C07313=1182.228,-66.696,-41.823,179.386,5.709,149.194
C07314=1182.223,-66.447,-41.834,179.389,5.710,149.194
C07315=1182.217,-66.196,-41.845,179.392,5.710,149.193
C07316=1182.213,-65.947,-41.856,179.393,5.710,149.192
C07317=1182.207,-65.697,-41.867,179.396,5.710,149.192
C07318=1182.202,-65.447,-41.878,179.398,5.711,149.191
C07319=1182.196,-65.198,-41.889,179.400,5.711,149.190
C07320=1182.191,-64.948,-41.900,179.403,5.711,149.190
C07321=1182.187,-64.698,-41.911,179.405,5.712,149.189
C07322=1182.181,-64.449,-41.921,179.407,5.712,149.189
C07323=1182.176,-64.199,-41.933,179.410,5.712,149.188
C07324=1182.171,-63.949,-41.945,179.412,5.713,149.187
C07325=1182.165,-63.700,-41.955,179.415,5.713,149.187
C07326=1182.161,-63.450,-41.966,179.417,5.713,149.186
C07327=1182.155,-63.200,-41.978,179.419,5.714,149.185
C07328=1182.150,-62.951,-41.988,179.422,5.714,149.185
C07329=1182.145,-62.701,-41.999,179.424,5.714,149.184
C07330=1182.139,-62.451,-42.011,179.426,5.715,149.184
C07331=1182.134,-62.201,-42.022,179.429,5.715,149.183
C07332=1182.129,-61.952,-42.033,179.431,5.715,149.182
C07333=1182.124,-61.702,-42.045,179.433,5.715,149.182
C07334=1182.118,-61.452,-42.055,179.436,5.716,149.181
C07335=1182.113,-61.203,-42.066,179.438,5.716,149.180
C07336=1182.108,-60.953,-42.078,179.440,5.716,149.180
C07337=1182.102,-60.703,-42.088,179.442,5.717,149.179
C07338=1182.098,-60.454,-42.100,179.445,5.717,149.178
C07339=1182.092,-60.204,-42.112,179.447,5.717,149.178
C07340=1182.087,-59.955,-42.122,179.449,5.718,149.177
C07341=1182.082,-59.705,-42.133,179.452,5.718,149.177
C07342=1182.077,-59.455,-42.145,179.454,5.718,149.176
C07343=1182.072,-59.205,-42.156,179.456,5.718,149.175
C07344=1182.067,-58.956,-42.167,179.459,5.719,149.175
C07345=1182.061,-58.705,-42.178,179.461,5.719,149.174
C07346=1182.056,-58.456,-42.190,179.463,5.719,149.173
C07347=1182.051,-58.206,-42.201,179.466,5.720,149.173
C07348=1182.045,-57.957,-42.212,179.468,5.721,149.172
C07349=1182.041,-57.707,-42.224,179.470,5.720,149.172
C07350=1182.035,-57.457,-42.235,179.473,5.721,149.171
C07351=1182.030,-57.208,-42.246,179.475,5.721,149.170
C07352=1182.024,-56.958,-42.258,179.477,5.721,149.170
C07353=1182.020,-56.708,-42.269,179.480,5.721,149.169
C07354=1182.015,-56.459,-42.280,179.482,5.722,149.169
C07355=1182.009,-56.209,-42.292,179.485,5.723,149.168
C07356=1182.004,-55.959,-42.302,179.487,5.722,149.167
C07357=1181.998,-55.709,-42.314,179.489,5.723,149.167
C07358=1181.994,-55.460,-42.325,179.492,5.724,149.166
C07359=1181.988,-55.210,-42.337,179.494,5.723,149.165
C07360=1181.983,-54.961,-42.348,179.496,5.724,149.165
C07361=1181.978,-54.711,-42.360,179.498,5.724,149.164
C07362=1181.973,-54.461,-42.371,179.501,5.725,149.163
C07363=1181.967,-54.211,-42.383,179.503,5.725,149.163
C07364=1181.963,-53.962,-42.395,179.505,5.725,149.162
C07365=1181.956,-53.712,-42.405,179.508,5.726,149.161
C07366=1181.952,-53.462,-42.417,179.511,5.726,149.161
C07367=1181.947,-53.213,-42.428,179.512,5.726,149.160
C07368=1181.942,-52.963,-42.440,179.515,5.727,149.160
C07369=1181.936,-52.713,-42.452,179.518,5.727,149.159
C07370=1181.931,-52.464,-42.463,179.519,5.727,149.158
C07371=1181.925,-52.214,-42.475,179.522,5.727,149.158
C07372=1181.921,-51.964,-42.486,179.525,5.728,149.157
C07373=1181.915,-51.714,-42.498,179.527,5.729,149.157
C07374=1181.911,-51.465,-42.509,179.529,5.728,149.156
C07375=1181.905,-51.215,-42.521,179.532,5.729,149.155
C07376=1181.900,-50.966,-42.532,179.534,5.730,149.155
C07377=1181.894,-50.716,-42.544,179.536,5.730,149.154
C07378=1181.890,-50.466,-42.555,179.538,5.730,149.153
C07379=1181.884,-50.216,-42.567,179.541,5.730,149.153
C07380=1181.878,-49.947,-42.580,179.543,5.731,149.152
C07381=1181.873,-49.676,-42.592,179.546,5.731,149.151
C07382=1181.868,-49.405,-42.605,179.549,5.732,149.151
C07383=1181.862,-49.136,-42.617,179.551,5.732,149.150
C07384=1181.857,-48.886,-42.629,179.553,5.732,149.149
C07385=1181.851,-48.636,-42.641,179.556,5.733,149.149
C07386=1181.846,-48.386,-42.652,179.558,5.733,149.148
C07387=1181.841,-48.137,-42.664,179.561,5.733,149.147
C07388=1181.836,-47.887,-42.676,179.562,5.733,149.147
C07389=1181.830,-47.637,-42.687,179.565,5.734,149.146
C07390=1181.825,-47.388,-42.698,179.568,5.734,149.145
C07391=1181.820,-47.138,-42.710,179.570,5.735,149.145
C07392=1181.815,-46.888,-42.722,179.572,5.735,149.144
C07393=1181.810,-46.639,-42.734,179.575,5.735,149.144
C07394=1181.805,-46.389,-42.746,179.577,5.736,149.143
C07395=1181.800,-46.139,-42.757,179.580,5.736,149.142
C07396=1181.794,-45.889,-42.769,179.582,5.737,149.142
C07397=1181.789,-45.639,-42.781,179.584,5.737,149.141
C07398=1181.784,-45.390,-42.792,179.587,5.737,149.141
C07399=1181.779,-45.141,-42.805,179.589,5.738,149.140
C07400=1181.773,-44.891,-42.817,179.592,5.738,149.139
C07401=1181.768,-44.642,-42.828,179.593,5.738,149.139
C07402=1181.763,-44.392,-42.840,179.596,5.739,149.138
C07403=1181.758,-44.142,-42.852,179.599,5.739,149.137
C07404=1181.752,-43.892,-42.864,179.601,5.740,149.137
C07405=1181.748,-43.643,-42.876,179.603,5.740,149.136
C07406=1181.742,-43.393,-42.887,179.606,5.740,149.135
C07407=1181.737,-43.143,-42.899,179.608,5.741,149.135
C07408=1181.732,-42.893,-42.911,179.611,5.741,149.134
C07409=1181.727,-42.644,-42.923,179.613,5.741,149.134
C07410=1181.722,-42.394,-42.935,179.615,5.741,149.133
C07411=1181.716,-42.144,-42.947,179.617,5.742,149.132
C07412=1181.712,-41.894,-42.958,179.620,5.743,149.132
C07413=1181.706,-41.645,-42.971,179.623,5.743,149.131
C07414=1181.701,-41.395,-42.983,179.624,5.743,149.130
C07415=1181.696,-41.145,-42.995,179.627,5.743,149.130
C07416=1181.691,-40.896,-43.007,179.630,5.744,149.129
C07417=1181.686,-40.646,-43.018,179.632,5.745,149.129
C07418=1181.680,-40.396,-43.030,179.635,5.745,149.128
C07419=1181.675,-40.147,-43.043,179.637,5.745,149.127
C07420=1181.670,-39.897,-43.055,179.639,5.745,149.126
C07421=1181.664,-39.648,-43.066,179.641,5.746,149.126
C07422=1181.659,-39.399,-43.078,179.644,5.746,149.125
C07423=1181.654,-39.149,-43.090,179.646,5.746,149.125
C07424=1181.648,-38.899,-43.102,179.648,5.747,149.124
C07425=1181.643,-38.650,-43.115,179.651,5.747,149.123
C07426=1181.639,-38.400,-43.126,179.654,5.748,149.123
C07427=1181.633,-38.150,-43.138,179.656,5.749,149.122
C07428=1181.628,-37.901,-43.151,179.658,5.748,149.122
C07429=1181.623,-37.650,-43.163,179.661,5.749,149.121
C07430=1181.618,-37.401,-43.175,179.663,5.750,149.120
C07431=1181.613,-37.151,-43.187,179.665,5.750,149.120
C07432=1181.608,-36.901,-43.199,179.668,5.750,149.119
C07433=1181.603,-36.652,-43.211,179.670,5.750,149.118
C07434=1181.597,-36.402,-43.223,179.672,5.751,149.118
C07435=1181.592,-36.153,-43.236,179.675,5.751,149.117
C07436=1181.587,-35.903,-43.248,179.678,5.752,149.116
C07437=1181.582,-35.653,-43.260,179.680,5.753,149.116
C07438=1181.576,-35.404,-43.272,179.682,5.752,149.115
C07439=1181.571,-35.154,-43.285,179.685,5.753,149.115
C07440=1181.566,-34.904,-43.296,179.687,5.753,149.114
C07441=1181.561,-34.655,-43.309,179.689,5.754,149.113
C07442=1181.556,-34.405,-43.320,179.692,5.754,149.113
C07443=1181.551,-34.156,-43.333,179.695,5.755,149.112
C07444=1181.545,-33.906,-43.345,179.696,5.755,149.112
C07445=1181.540,-33.657,-43.357,179.699,5.755,149.111
C07446=1181.535,-33.407,-43.369,179.702,5.756,149.110
C07447=1181.530,-33.158,-43.382,179.704,5.757,149.110
C07448=1181.525,-32.907,-43.394,179.707,5.757,149.109
C07449=1181.520,-32.658,-43.407,179.709,5.757,149.108
C07450=1181.514,-32.408,-43.419,179.711,5.757,149.108
C07451=1181.509,-32.158,-43.431,179.713,5.758,149.107
C07452=1181.504,-31.908,-43.443,179.716,5.758,149.106
C07453=1181.499,-31.659,-43.456,179.719,5.759,149.106
C07454=1181.494,-31.410,-43.468,179.721,5.760,149.105
C07455=1181.488,-31.160,-43.480,179.723,5.759,149.105
C07456=1181.483,-30.910,-43.493,179.726,5.760,149.104
C07457=1181.478,-30.660,-43.505,179.728,5.761,149.103
C07458=1181.473,-30.411,-43.518,179.731,5.761,149.103
C07459=1181.468,-30.161,-43.530,179.733,5.761,149.102
C07460=1181.463,-29.911,-43.542,179.735,5.762,149.101
C07461=1181.457,-29.662,-43.555,179.737,5.762,149.101
C07462=1181.452,-29.413,-43.567,179.740,5.762,149.100
C07463=1181.447,-29.163,-43.579,179.743,5.763,149.099
C07464=1181.442,-28.913,-43.592,179.745,5.764,149.099
C07465=1181.437,-28.663,-43.605,179.748,5.764,149.098
C07466=1181.432,-28.413,-43.617,179.750,5.764,149.098
C07467=1181.427,-28.164,-43.629,179.752,5.765,149.097
C07468=1181.422,-27.915,-43.642,179.755,5.765,149.096
C07469=1181.416,-27.665,-43.654,179.757,5.765,149.096
C07470=1181.412,-27.415,-43.667,179.759,5.766,149.095
C07471=1181.406,-27.166,-43.679,179.762,5.767,149.094
C07472=1181.401,-26.916,-43.692,179.765,5.767,149.094
C07473=1181.396,-26.666,-43.704,179.767,5.767,149.093
C07474=1181.391,-26.417,-43.716,179.769,5.768,149.093
C07475=1181.386,-26.168,-43.729,179.772,5.768,149.092
C07476=1181.381,-25.918,-43.742,179.774,5.769,149.091
C07477=1181.375,-25.667,-43.755,179.776,5.769,149.091
C07478=1181.370,-25.418,-43.767,179.779,5.770,149.090
C07479=1181.365,-25.169,-43.780,179.782,5.770,149.089
C07480=1181.360,-24.919,-43.792,179.783,5.770,149.089
C07481=1181.355,-24.669,-43.805,179.786,5.771,149.088
C07482=1181.350,-24.419,-43.817,179.789,5.771,149.087
C07483=1181.345,-24.170,-43.830,179.791,5.772,149.087
C07484=1181.339,-23.900,-43.844,179.794,5.772,149.086
C07485=1181.333,-23.631,-43.857,179.796,5.773,149.086
C07486=1181.328,-23.361,-43.871,179.799,5.773,149.085
C07487=1181.322,-23.091,-43.885,179.801,5.774,149.084
C07488=1181.317,-22.841,-43.897,179.804,5.774,149.084
C07489=1181.312,-22.592,-43.910,179.807,5.775,149.083
C07490=1181.307,-22.343,-43.922,179.809,5.776,149.082
C07491=1181.301,-22.092,-43.936,179.812,5.776,149.082
C07492=1181.296,-21.843,-43.949,179.814,5.776,149.081
C07493=1181.291,-21.594,-43.961,179.816,5.776,149.081
C07494=1181.286,-21.344,-43.974,179.819,5.777,149.080
C07495=1181.282,-21.094,-43.987,179.821,5.777,149.079
C07496=1181.275,-20.844,-43.999,179.824,5.778,149.078
C07497=1181.270,-20.595,-44.012,179.826,5.779,149.078
C07498=1181.266,-20.345,-44.025,179.829,5.779,149.077
C07499=1181.261,-20.096,-44.037,179.831,5.780,149.077
C07500=1181.255,-19.846,-44.051,179.833,5.780,149.076
C07501=1181.250,-19.597,-44.063,179.836,5.780,149.075
C07502=1181.245,-19.347,-44.076,179.838,5.781,149.075
C07503=1181.240,-19.097,-44.089,179.841,5.781,149.074
C07504=1181.234,-18.848,-44.102,179.843,5.782,149.074
C07505=1181.230,-18.598,-44.115,179.846,5.782,149.073
C07506=1181.225,-18.348,-44.128,179.848,5.783,149.072
C07507=1181.219,-18.099,-44.140,179.851,5.784,149.072
C07508=1181.214,-17.849,-44.153,179.853,5.783,149.071
C07509=1181.209,-17.599,-44.166,179.855,5.784,149.070
C07510=1181.204,-17.350,-44.179,179.858,5.784,149.070
C07511=1181.199,-17.101,-44.191,179.860,5.785,149.069
C07512=1181.194,-16.850,-44.205,179.863,5.785,149.068
C07513=1181.188,-16.601,-44.218,179.865,5.786,149.068
C07514=1181.183,-16.352,-44.230,179.868,5.787,149.067
C07515=1181.178,-16.101,-44.244,179.870,5.787,149.067
C07516=1181.173,-15.852,-44.256,179.873,5.788,149.066
C07517=1181.168,-15.603,-44.270,179.875,5.788,149.065
C07518=1181.163,-15.353,-44.283,179.877,5.788,149.065
C07519=1181.158,-15.104,-44.296,179.880,5.789,149.064
C07520=1181.153,-14.854,-44.309,179.882,5.789,149.064
C07521=1181.147,-14.604,-44.322,179.885,5.790,149.063
C07522=1181.142,-14.355,-44.335,179.887,5.790,149.062
C07523=1181.138,-14.105,-44.348,179.890,5.791,149.062
C07524=1181.132,-13.855,-44.361,179.892,5.792,149.061
C07525=1181.127,-13.606,-44.374,179.895,5.792,149.060
C07526=1181.122,-13.356,-44.388,179.898,5.793,149.060
C07527=1181.117,-13.107,-44.400,179.900,5.793,149.059
C07528=1181.112,-12.857,-44.413,179.902,5.794,149.059
C07529=1181.106,-12.607,-44.426,179.904,5.793,149.058
C07530=1181.101,-12.358,-44.439,179.907,5.794,149.057
C07531=1181.097,-12.108,-44.453,179.909,5.795,149.057
C07532=1181.091,-11.859,-44.466,179.912,5.795,149.056
C07533=1181.086,-11.609,-44.479,179.915,5.796,149.055
C07534=1181.081,-11.359,-44.492,179.917,5.797,149.055
C07535=1181.076,-11.110,-44.505,179.919,5.797,149.054
C07536=1181.071,-10.860,-44.519,179.922,5.797,149.053
C07537=1181.065,-10.611,-44.532,179.924,5.798,149.053
C07538=1181.061,-10.361,-44.545,179.927,5.799,149.052
C07539=1181.055,-10.112,-44.558,179.930,5.799,149.052
C07540=1181.051,-9.862,-44.571,179.932,5.800,149.051
C07541=1181.045,-9.612,-44.585,179.934,5.800,149.050
C07542=1181.040,-9.363,-44.597,179.936,5.800,149.050
C07543=1181.035,-9.113,-44.612,179.939,5.801,149.049
C07544=1181.030,-8.864,-44.624,179.941,5.801,149.049
C07545=1181.024,-8.613,-44.638,179.944,5.802,149.048
C07546=1181.020,-8.365,-44.651,179.947,5.802,149.047
C07547=1181.014,-8.114,-44.665,179.949,5.803,149.047
C07548=1181.009,-7.865,-44.677,179.951,5.804,149.046
C07549=1181.004,-7.615,-44.691,179.954,5.804,149.045
C07550=1180.999,-7.366,-44.704,179.956,5.805,149.045
C07551=1180.994,-7.116,-44.718,179.959,5.805,149.044
C07552=1180.989,-6.867,-44.731,179.962,5.806,149.043
C07553=1180.984,-6.617,-44.744,179.964,5.806,149.043
C07554=1180.979,-6.367,-44.757,179.966,5.807,149.042
C07555=1180.974,-6.118,-44.771,179.969,5.808,149.042
C07556=1180.969,-5.868,-44.784,179.972,5.808,149.041
C07557=1180.964,-5.619,-44.798,179.974,5.809,149.040
C07558=1180.959,-5.369,-44.811,179.977,5.809,149.040
C07559=1180.953,-5.119,-44.824,179.979,5.810,149.039
C07560=1180.948,-4.870,-44.838,179.981,5.810,149.039
C07561=1180.943,-4.620,-44.851,179.983,5.810,149.038
C07562=1180.938,-4.371,-44.865,179.986,5.811,149.037
C07563=1180.933,-4.121,-44.878,179.989,5.811,149.037
C07564=1180.928,-3.872,-44.892,179.991,5.812,149.036
C07565=1180.922,-3.622,-44.906,179.994,5.813,149.035
C07566=1180.918,-3.373,-44.919,179.996,5.813,149.035
C07567=1180.912,-3.123,-44.932,179.998,5.814,149.034
C07568=1180.907,-2.874,-44.946,-179.999,5.814,149.034
C07569=1180.902,-2.624,-44.959,-179.996,5.815,149.033
C07570=1180.897,-2.375,-44.973,-179.994,5.816,149.032
C07571=1180.892,-2.125,-44.986,-179.992,5.816,149.032
C07572=1180.887,-1.875,-45.001,-179.989,5.817,149.031
C07573=1180.881,-1.625,-45.014,-179.986,5.817,149.030
C07574=1180.877,-1.376,-45.027,-179.984,5.818,149.030
C07575=1180.871,-1.126,-45.041,-179.981,5.818,149.029
C07576=1180.866,-0.876,-45.055,-179.979,5.819,149.029
C07577=1180.861,-0.627,-45.067,-179.977,5.820,149.028
C07578=1180.856,-0.377,-45.082,-179.974,5.820,149.027
C07579=1180.851,-0.128,-45.096,-179.971,5.821,149.027
C07580=1180.846,0.122,-45.109,-179.969,5.822,149.026
C07581=1180.841,0.371,-45.123,-179.966,5.822,149.026
C07582=1180.835,0.621,-45.136,-179.964,5.823,149.025
C07583=1180.831,0.870,-45.150,-179.962,5.823,149.024
C07584=1180.826,1.119,-45.164,-179.959,5.824,149.024
C07585=1180.820,1.370,-45.177,-179.956,5.824,149.023
C07586=1180.815,1.619,-45.192,-179.954,5.825,149.022
C07587=1180.810,1.868,-45.205,-179.951,5.826,149.022
C07588=1180.805,2.138,-45.220,-179.949,5.826,149.021
C07589=1180.800,2.407,-45.235,-179.946,5.827,149.020
C07590=1180.794,2.676,-45.250,-179.943,5.827,149.020
C07591=1180.788,2.945,-45.264,-179.941,5.828,149.019
C07592=1180.783,3.195,-45.278,-179.938,5.828,149.018
C07593=1180.779,3.445,-45.292,-179.936,5.829,149.018
C07594=1180.773,3.694,-45.306,-179.933,5.829,149.017
C07595=1180.768,3.944,-45.319,-179.931,5.830,149.017
C07596=1180.763,4.194,-45.333,-179.929,5.831,149.016
C07597=1180.758,4.443,-45.347,-179.926,5.831,149.015
C07598=1180.753,4.692,-45.361,-179.923,5.832,149.015
C07599=1180.748,4.943,-45.375,-179.921,5.832,149.014
C07600=1180.742,5.192,-45.389,-179.918,5.833,149.014
C07601=1180.737,5.441,-45.403,-179.916,5.833,149.013
C07602=1180.733,5.691,-45.416,-179.914,5.834,149.012
C07603=1180.727,5.940,-45.430,-179.911,5.835,149.012
C07604=1180.722,6.190,-45.444,-179.908,5.835,149.011
C07605=1180.717,6.440,-45.458,-179.906,5.836,149.011
C07606=1180.712,6.689,-45.472,-179.903,5.836,149.010
C07607=1180.707,6.938,-45.486,-179.901,5.837,149.009
C07608=1180.703,7.188,-45.500,-179.898,5.837,149.009
C07609=1180.697,7.437,-45.513,-179.896,5.838,149.008
C07610=1180.692,7.687,-45.528,-179.893,5.840,149.007
C07611=1180.687,7.937,-45.542,-179.890,5.840,149.007
C07612=1180.682,8.187,-45.556,-179.888,5.841,149.006
C07613=1180.676,8.436,-45.570,-179.885,5.841,149.006
C07614=1180.671,8.685,-45.584,-179.883,5.842,149.005
C07615=1180.666,8.935,-45.599,-179.880,5.843,149.004
C07616=1180.661,9.184,-45.611,-179.878,5.843,149.004
C07617=1180.656,9.434,-45.625,-179.875,5.844,149.003
C07618=1180.651,9.684,-45.640,-179.873,5.845,149.003
C07619=1180.646,9.934,-45.654,-179.870,5.845,149.002
C07620=1180.641,10.183,-45.668,-179.868,5.845,149.001
C07621=1180.636,10.432,-45.682,-179.866,5.846,149.001
C07622=1180.631,10.682,-45.696,-179.863,5.847,149.000
C07623=1180.626,10.932,-45.711,-179.860,5.847,148.999
C07624=1180.620,11.181,-45.725,-179.858,5.848,148.999
C07625=1180.616,11.430,-45.739,-179.855,5.849,148.998
C07626=1180.611,11.680,-45.753,-179.853,5.849,148.998
C07627=1180.606,11.930,-45.767,-179.851,5.850,148.997
C07628=1180.601,12.179,-45.782,-179.848,5.850,148.996
C07629=1180.595,12.428,-45.796,-179.845,5.851,148.996
C07630=1180.590,12.678,-45.810,-179.843,5.851,148.995
C07631=1180.585,12.928,-45.824,-179.840,5.852,148.995
C07632=1180.580,13.178,-45.839,-179.838,5.853,148.994
C07633=1180.575,13.427,-45.852,-179.835,5.853,148.993
C07634=1180.570,13.676,-45.867,-179.833,5.854,148.993
C07635=1180.565,13.926,-45.881,-179.830,5.855,148.992
C07636=1180.560,14.176,-45.895,-179.828,5.855,148.991
C07637=1180.555,14.425,-45.910,-179.825,5.857,148.991
C07638=1180.549,14.674,-45.923,-179.822,5.857,148.990
C07639=1180.544,14.924,-45.938,-179.820,5.858,148.990
C07640=1180.540,15.173,-45.953,-179.817,5.858,148.989
C07641=1180.535,15.423,-45.967,-179.815,5.859,148.988
C07642=1180.530,15.673,-45.981,-179.812,5.859,148.988
C07643=1180.525,15.922,-45.996,-179.810,5.860,148.987
C07644=1180.519,16.171,-46.009,-179.807,5.861,148.987
C07645=1180.514,16.421,-46.024,-179.805,5.861,148.986
C07646=1180.509,16.671,-46.038,-179.803,5.862,148.986
C07647=1180.504,16.921,-46.052,-179.800,5.863,148.985
C07648=1180.500,17.170,-46.067,-179.797,5.863,148.984
C07649=1180.494,17.420,-46.082,-179.795,5.864,148.984
C07650=1180.489,17.669,-46.096,-179.792,5.864,148.983
C07651=1180.484,17.918,-46.110,-179.790,5.865,148.982
C07652=1180.479,18.168,-46.125,-179.787,5.867,148.982
C07653=1180.474,18.417,-46.140,-179.784,5.867,148.981
C07654=1180.469,18.667,-46.154,-179.782,5.868,148.981
C07655=1180.464,18.917,-46.168,-179.780,5.868,148.980
C07656=1180.459,19.166,-46.182,-179.777,5.869,148.979
C07657=1180.454,19.416,-46.197,-179.774,5.869,148.979
C07658=1180.449,19.665,-46.212,-179.772,5.870,148.978
C07659=1180.444,19.915,-46.227,-179.769,5.871,148.978
C07660=1180.438,20.164,-46.241,-179.767,5.871,148.977
C07661=1180.434,20.413,-46.255,-179.765,5.872,148.976
C07662=1180.429,20.663,-46.270,-179.762,5.873,148.976
C07663=1180.424,20.913,-46.284,-179.759,5.873,148.975
C07664=1180.418,21.163,-46.299,-179.757,5.875,148.975
C07665=1180.413,21.412,-46.314,-179.754,5.875,148.974
C07666=1180.408,21.662,-46.328,-179.751,5.876,148.973
C07667=1180.403,21.911,-46.342,-179.749,5.877,148.973
C07668=1180.399,22.160,-46.357,-179.747,5.877,148.972
C07669=1180.393,22.410,-46.372,-179.744,5.878,148.971
C07670=1180.388,22.660,-46.387,-179.742,5.878,148.971
C07671=1180.383,22.909,-46.402,-179.739,5.879,148.970
C07672=1180.379,23.159,-46.416,-179.736,5.879,148.970
C07673=1180.373,23.409,-46.431,-179.734,5.880,148.969
C07674=1180.368,23.657,-46.445,-179.731,5.882,148.968
C07675=1180.363,23.907,-46.460,-179.728,5.882,148.968
C07676=1180.358,24.156,-46.475,-179.726,5.883,148.967
C07677=1180.352,24.406,-46.490,-179.724,5.883,148.967
C07678=1180.348,24.655,-46.505,-179.721,5.884,148.966
C07679=1180.343,24.905,-46.519,-179.719,5.885,148.966
C07680=1180.338,25.155,-46.533,-179.716,5.885,148.965
C07681=1180.332,25.404,-46.549,-179.714,5.886,148.964
C07682=1180.327,25.654,-46.563,-179.711,5.887,148.964
C07683=1180.323,25.903,-46.578,-179.708,5.888,148.963
C07684=1180.317,26.153,-46.593,-179.706,5.889,148.963
C07685=1180.312,26.402,-46.608,-179.703,5.889,148.962
C07686=1180.307,26.652,-46.622,-179.701,5.890,148.961
C07687=1180.302,26.901,-46.638,-179.698,5.891,148.961
C07688=1180.297,27.151,-46.652,-179.696,5.891,148.960
C07689=1180.292,27.400,-46.667,-179.693,5.892,148.959
C07690=1180.287,27.650,-46.682,-179.691,5.892,148.959
C07691=1180.282,27.899,-46.697,-179.688,5.894,148.958
C07692=1180.277,28.168,-46.713,-179.685,5.894,148.958
C07693=1180.271,28.437,-46.729,-179.682,5.895,148.957
C07694=1180.266,28.706,-46.745,-179.679,5.896,148.956
C07695=1180.260,28.975,-46.761,-179.677,5.897,148.956
C07696=1180.255,29.224,-46.776,-179.674,5.897,148.955
C07697=1180.251,29.473,-46.791,-179.672,5.898,148.954
C07698=1180.245,29.723,-46.806,-179.670,5.899,148.954
C07699=1180.241,29.972,-46.821,-179.667,5.899,148.953
C07700=1180.235,30.223,-46.836,-179.664,5.900,148.953
C07701=1180.231,30.472,-46.851,-179.662,5.901,148.952
C07702=1180.226,30.721,-46.866,-179.659,5.902,148.952
C07703=1180.220,30.971,-46.881,-179.656,5.902,148.951
C07704=1180.216,31.220,-46.896,-179.654,5.903,148.950
C07705=1180.210,31.469,-46.911,-179.652,5.904,148.950
C07706=1180.205,31.719,-46.926,-179.649,5.905,148.949
C07707=1180.200,31.969,-46.941,-179.646,5.906,148.949
C07708=1180.195,32.218,-46.956,-179.643,5.906,148.948
C07709=1180.190,32.468,-46.971,-179.641,5.907,148.947
C07710=1180.185,32.717,-46.986,-179.639,5.908,148.947
C07711=1180.181,32.967,-47.001,-179.636,5.908,148.946
C07712=1180.175,33.217,-47.016,-179.634,5.909,148.946
C07713=1180.171,33.466,-47.031,-179.631,5.910,148.945
C07714=1180.165,33.715,-47.047,-179.628,5.911,148.944
C07715=1180.161,33.964,-47.062,-179.626,5.912,148.944
C07716=1180.155,34.214,-47.077,-179.623,5.912,148.943
C07717=1180.150,34.463,-47.092,-179.621,5.913,148.943
C07718=1180.145,34.713,-47.107,-179.618,5.914,148.942
C07719=1180.140,34.963,-47.123,-179.615,5.915,148.941
C07720=1180.135,35.212,-47.138,-179.613,5.916,148.941
C07721=1180.130,35.462,-47.153,-179.610,5.916,148.940
C07722=1180.125,35.711,-47.168,-179.608,5.917,148.940
C07723=1180.120,35.960,-47.184,-179.606,5.918,148.939
C07724=1180.115,36.209,-47.199,-179.603,5.918,148.938
C07725=1180.110,36.459,-47.214,-179.600,5.919,148.938
C07726=1180.105,36.709,-47.229,-179.598,5.920,148.937
C07727=1180.100,36.959,-47.245,-179.595,5.921,148.937
C07728=1180.095,37.208,-47.260,-179.593,5.922,148.936
C07729=1180.090,37.457,-47.275,-179.590,5.922,148.936
C07730=1180.085,37.707,-47.291,-179.587,5.923,148.935
C07731=1180.080,37.956,-47.306,-179.585,5.924,148.934
C07732=1180.075,38.206,-47.322,-179.582,5.925,148.934
C07733=1180.070,38.455,-47.337,-179.579,5.925,148.933
C07734=1180.065,38.705,-47.352,-179.577,5.926,148.933
C07735=1180.059,38.954,-47.367,-179.575,5.927,148.932
C07736=1180.055,39.203,-47.382,-179.572,5.928,148.932
C07737=1180.050,39.453,-47.398,-179.569,5.929,148.931
C07738=1180.045,39.703,-47.414,-179.567,5.929,148.930
C07739=1180.040,39.952,-47.429,-179.564,5.930,148.930
C07740=1180.035,40.201,-47.444,-179.562,5.931,148.929
C07741=1180.030,40.451,-47.460,-179.559,5.932,148.929
C07742=1180.025,40.701,-47.475,-179.556,5.933,148.928
C07743=1180.020,40.950,-47.491,-179.554,5.933,148.927
C07744=1180.014,41.199,-47.506,-179.552,5.934,148.927
C07745=1180.010,41.448,-47.521,-179.549,5.935,148.926
C07746=1180.005,41.699,-47.537,-179.546,5.936,148.926
C07747=1179.999,41.948,-47.553,-179.544,5.937,148.925
C07748=1179.995,42.197,-47.568,-179.541,5.938,148.924
C07749=1179.990,42.447,-47.584,-179.539,5.938,148.924
C07750=1179.985,42.697,-47.599,-179.536,5.940,148.923
C07751=1179.979,42.946,-47.615,-179.533,5.940,148.923
C07752=1179.975,43.195,-47.630,-179.531,5.941,148.922
C07753=1179.970,43.445,-47.646,-179.528,5.942,148.921
C07754=1179.965,43.694,-47.662,-179.526,5.943,148.921
C07755=1179.959,43.943,-47.678,-179.523,5.944,148.920
C07756=1179.955,44.192,-47.693,-179.520,5.944,148.920
C07757=1179.950,44.443,-47.709,-179.518,5.945,148.919
C07758=1179.945,44.692,-47.724,-179.515,5.946,148.919
C07759=1179.939,44.941,-47.740,-179.513,5.947,148.918
C07760=1179.935,45.191,-47.755,-179.510,5.948,148.917
C07761=1179.930,45.441,-47.771,-179.507,5.948,148.917
C07762=1179.925,45.689,-47.787,-179.505,5.949,148.916
C07763=1179.920,45.939,-47.803,-179.503,5.950,148.916
C07764=1179.914,46.189,-47.819,-179.499,5.951,148.915
C07765=1179.910,46.438,-47.834,-179.497,5.952,148.915
C07766=1179.905,46.688,-47.850,-179.495,5.952,148.914
C07767=1179.900,46.937,-47.866,-179.492,5.953,148.913
C07768=1179.895,47.186,-47.882,-179.489,5.955,148.913
C07769=1179.890,47.436,-47.898,-179.486,5.955,148.912
C07770=1179.885,47.685,-47.913,-179.484,5.956,148.912
C07771=1179.880,47.934,-47.929,-179.482,5.957,148.911
C07772=1179.875,48.184,-47.945,-179.479,5.958,148.911
C07773=1179.870,48.434,-47.960,-179.476,5.959,148.910
C07774=1179.864,48.683,-47.976,-179.474,5.960,148.909
C07775=1179.860,48.933,-47.993,-179.472,5.960,148.909
C07776=1179.855,49.182,-48.008,-179.468,5.961,148.908
C07777=1179.851,49.432,-48.024,-179.466,5.962,148.908
C07778=1179.845,49.681,-48.039,-179.464,5.963,148.907
C07779=1179.840,49.930,-48.055,-179.461,5.964,148.907
C07780=1179.835,50.180,-48.071,-179.458,5.965,148.906
C07781=1179.830,50.429,-48.087,-179.456,5.966,148.905
C07782=1179.825,50.679,-48.104,-179.453,5.966,148.905
C07783=1179.820,50.928,-48.119,-179.451,5.967,148.904
C07784=1179.815,51.177,-48.136,-179.448,5.969,148.904
C07785=1179.810,51.427,-48.152,-179.445,5.969,148.903
C07786=1179.805,51.677,-48.167,-179.443,5.970,148.902
C07787=1179.800,51.926,-48.184,-179.440,5.971,148.902
C07788=1179.795,52.176,-48.199,-179.437,5.972,148.901
C07789=1179.791,52.424,-48.215,-179.435,5.973,148.901
C07790=1179.786,52.674,-48.231,-179.433,5.973,148.900
C07791=1179.780,52.924,-48.247,-179.430,5.975,148.900
C07792=1179.776,53.173,-48.263,-179.427,5.975,148.899
C07793=1179.771,53.422,-48.279,-179.425,5.976,148.898
C07794=1179.766,53.672,-48.296,-179.422,5.977,148.898
C07795=1179.761,53.921,-48.311,-179.419,5.978,148.897
C07796=1179.755,54.190,-48.328,-179.417,5.979,148.897
C07797=1179.750,54.459,-48.347,-179.414,5.980,148.896
C07798=1179.744,54.727,-48.364,-179.411,5.981,148.895
C07799=1179.739,54.996,-48.381,-179.408,5.982,148.895
C07800=1179.734,55.245,-48.398,-179.406,5.983,148.894
C07801=1179.729,55.494,-48.413,-179.403,5.984,148.894
C07802=1179.724,55.744,-48.430,-179.401,5.984,148.893
C07803=1179.719,55.993,-48.445,-179.398,5.986,148.893
C07804=1179.714,56.243,-48.462,-179.395,5.986,148.892
C07805=1179.709,56.492,-48.478,-179.393,5.987,148.892
C07806=1179.705,56.742,-48.494,-179.390,5.989,148.891
C07807=1179.699,56.991,-48.511,-179.388,5.989,148.890
C07808=1179.695,57.241,-48.527,-179.385,5.990,148.890
C07809=1179.690,57.489,-48.543,-179.382,5.991,148.889
C07810=1179.685,57.740,-48.559,-179.380,5.992,148.889
C07811=1179.679,57.989,-48.576,-179.377,5.993,148.888
C07812=1179.675,58.238,-48.592,-179.375,5.994,148.888
C07813=1179.669,58.487,-48.608,-179.372,5.995,148.887
C07814=1179.665,58.737,-48.625,-179.369,5.996,148.886
C07815=1179.659,58.986,-48.640,-179.367,5.996,148.886
C07816=1179.655,59.236,-48.657,-179.364,5.998,148.885
C07817=1179.650,59.485,-48.673,-179.361,5.998,148.885
C07818=1179.645,59.735,-48.689,-179.359,5.999,148.884
C07819=1179.639,59.984,-48.706,-179.356,6.001,148.884
C07820=1179.635,60.233,-48.723,-179.353,6.001,148.883
C07821=1179.630,60.483,-48.739,-179.351,6.002,148.882
C07822=1179.625,60.732,-48.755,-179.348,6.003,148.882
C07823=1179.620,60.982,-48.772,-179.346,6.004,148.881
C07824=1179.615,61.230,-48.788,-179.343,6.005,148.881
C07825=1179.610,61.481,-48.805,-179.341,6.007,148.880
C07826=1179.605,61.730,-48.821,-179.338,6.007,148.880
C07827=1179.600,61.979,-48.837,-179.335,6.008,148.879
C07828=1179.596,62.229,-48.854,-179.333,6.009,148.879
C07829=1179.590,62.478,-48.870,-179.330,6.010,148.878
C07830=1179.585,62.728,-48.887,-179.328,6.011,148.877
C07831=1179.580,62.977,-48.903,-179.325,6.012,148.877
C07832=1179.575,63.226,-48.920,-179.322,6.013,148.876
C07833=1179.571,63.476,-48.937,-179.320,6.013,148.876
C07834=1179.565,63.725,-48.953,-179.317,6.015,148.875
C07835=1179.560,63.975,-48.970,-179.314,6.016,148.875
C07836=1179.556,64.224,-48.986,-179.312,6.017,148.874
C07837=1179.551,64.473,-49.002,-179.309,6.018,148.873
C07838=1179.546,64.723,-49.020,-179.306,6.018,148.873
C07839=1179.541,64.972,-49.036,-179.304,6.019,148.872
C07840=1179.536,65.221,-49.053,-179.301,6.021,148.872
C07841=1179.531,65.471,-49.070,-179.299,6.021,148.871
C07842=1179.525,65.720,-49.086,-179.296,6.022,148.871
C07843=1179.521,65.970,-49.102,-179.294,6.024,148.870
C07844=1179.516,66.219,-49.119,-179.291,6.024,148.870
C07845=1179.511,66.468,-49.136,-179.288,6.026,148.869
C07846=1179.506,66.718,-49.152,-179.286,6.026,148.868
C07847=1179.502,66.967,-49.169,-179.283,6.027,148.868
C07848=1179.496,67.216,-49.186,-179.280,6.029,148.867
C07849=1179.491,67.466,-49.203,-179.278,6.030,148.867
C07850=1179.487,67.715,-49.219,-179.275,6.030,148.866
C07851=1179.482,67.965,-49.237,-179.273,6.032,148.866
C07852=1179.477,68.214,-49.253,-179.270,6.032,148.865
C07853=1179.471,68.464,-49.270,-179.268,6.033,148.865
C07854=1179.467,68.713,-49.287,-179.265,6.035,148.864
C07855=1179.462,68.962,-49.303,-179.262,6.035,148.863
C07856=1179.457,69.212,-49.320,-179.259,6.037,148.863
C07857=1179.452,69.461,-49.337,-179.257,6.037,148.862
C07858=1179.448,69.711,-49.354,-179.255,6.038,148.862
C07859=1179.442,69.960,-49.371,-179.251,6.040,148.861
C07860=1179.437,70.209,-49.387,-179.249,6.040,148.861
C07861=1179.432,70.459,-49.405,-179.247,6.041,148.860
C07862=1179.427,70.708,-49.421,-179.244,6.043,148.860
C07863=1179.422,70.958,-49.438,-179.241,6.043,148.859
C07864=1179.418,71.207,-49.456,-179.238,6.045,148.859
C07865=1179.413,71.456,-49.472,-179.236,6.045,148.858
C07866=1179.407,71.705,-49.489,-179.234,6.046,148.858
C07867=1179.403,71.955,-49.506,-179.231,6.048,148.857
C07868=1179.398,72.204,-49.523,-179.228,6.049,148.856
C07869=1179.393,72.454,-49.540,-179.225,6.050,148.856
C07870=1179.387,72.703,-49.557,-179.223,6.051,148.855
C07871=1179.383,72.952,-49.574,-179.220,6.051,148.855
C07872=1179.378,73.202,-49.591,-179.218,6.053,148.854
C07873=1179.374,73.451,-49.608,-179.215,6.054,148.854
C07874=1179.368,73.701,-49.625,-179.212,6.055,148.853
C07875=1179.363,73.950,-49.642,-179.210,6.056,148.853
C07876=1179.358,74.199,-49.660,-179.208,6.057,148.852
C07877=1179.354,74.448,-49.676,-179.204,6.058,148.851
C07878=1179.349,74.698,-49.693,-179.202,6.059,148.851
C07879=1179.344,74.948,-49.710,-179.199,6.060,148.850
C07880=1179.339,75.196,-49.728,-179.197,6.061,148.850
C07881=1179.333,75.446,-49.745,-179.194,6.062,148.849
C07882=1179.329,75.695,-49.762,-179.191,6.063,148.849
C07883=1179.324,75.945,-49.779,-179.189,6.064,148.848
C07884=1179.320,76.194,-49.796,-179.186,6.066,148.848
C07885=1179.314,76.444,-49.814,-179.183,6.066,148.847
C07886=1179.309,76.693,-49.830,-179.181,6.068,148.847
C07887=1179.304,76.942,-49.848,-179.178,6.068,148.846
C07888=1179.299,77.192,-49.865,-179.176,6.069,148.846
C07889=1179.295,77.441,-49.882,-179.173,6.071,148.845
C07890=1179.290,77.690,-49.900,-179.171,6.071,148.845
C07891=1179.285,77.940,-49.916,-179.167,6.073,148.844
C07892=1179.279,78.189,-49.933,-179.165,6.074,148.843
C07893=1179.274,78.438,-49.951,-179.162,6.075,148.843
C07894=1179.270,78.688,-49.968,-179.160,6.076,148.842
C07895=1179.265,78.937,-49.986,-179.157,6.077,148.842
C07896=1179.260,79.187,-50.003,-179.155,6.078,148.841
C07897=1179.255,79.436,-50.020,-179.152,6.079,148.841
C07898=1179.250,79.685,-50.038,-179.149,6.080,148.840
C07899=1179.245,79.935,-50.055,-179.147,6.081,148.840
C07900=1179.240,80.202,-50.074,-179.144,6.083,148.839
C07901=1179.235,80.471,-50.092,-179.141,6.083,148.838
C07902=1179.230,80.740,-50.111,-179.138,6.085,148.838
C07903=1179.224,81.008,-50.130,-179.135,6.086,148.837
C07904=1179.219,81.257,-50.147,-179.133,6.087,148.837
C07905=1179.214,81.506,-50.165,-179.130,6.089,148.836
C07906=1179.209,81.756,-50.182,-179.127,6.089,148.836
C07907=1179.204,82.005,-50.200,-179.125,6.091,148.835
C07908=1179.200,82.255,-50.217,-179.122,6.091,148.835
C07909=1179.195,82.504,-50.235,-179.120,6.092,148.834
C07910=1179.190,82.754,-50.252,-179.117,6.094,148.834
C07911=1179.185,83.003,-50.270,-179.114,6.094,148.833
C07912=1179.180,83.252,-50.286,-179.112,6.096,148.833
C07913=1179.175,83.501,-50.304,-179.109,6.097,148.832
C07914=1179.171,83.751,-50.322,-179.106,6.098,148.832
C07915=1179.165,84.000,-50.340,-179.104,6.099,148.831
C07916=1179.160,84.250,-50.358,-179.101,6.101,148.831
C07917=1179.156,84.499,-50.374,-179.098,6.101,148.830
C07918=1179.151,84.748,-50.392,-179.096,6.103,148.829
C07919=1179.146,84.997,-50.410,-179.093,6.103,148.829
C07920=1179.141,85.247,-50.428,-179.090,6.105,148.828
C07921=1179.136,85.496,-50.446,-179.088,6.106,148.828
C07922=1179.132,85.745,-50.463,-179.085,6.107,148.827
C07923=1179.127,85.995,-50.480,-179.083,6.108,148.827
C07924=1179.122,86.244,-50.498,-179.080,6.110,148.826
C07925=1179.117,86.493,-50.516,-179.078,6.111,148.826
C07926=1179.112,86.743,-50.533,-179.075,6.111,148.825
C07927=1179.107,86.992,-50.551,-179.072,6.113,148.825
C07928=1179.102,87.242,-50.569,-179.070,6.113,148.824
C07929=1179.097,87.491,-50.586,-179.067,6.115,148.824
C07930=1179.092,87.740,-50.604,-179.065,6.116,148.823
C07931=1179.087,87.989,-50.622,-179.062,6.117,148.823
C07932=1179.082,88.239,-50.640,-179.059,6.118,148.822
C07933=1179.077,88.488,-50.657,-179.056,6.120,148.822
C07934=1179.072,88.738,-50.675,-179.054,6.121,148.821
C07935=1179.067,88.987,-50.693,-179.051,6.122,148.820
C07936=1179.063,89.236,-50.711,-179.049,6.123,148.820
C07937=1179.058,89.485,-50.729,-179.045,6.124,148.819
C07938=1179.052,89.735,-50.746,-179.043,6.125,148.819
C07939=1179.047,89.984,-50.764,-179.041,6.127,148.819
C07940=1179.043,90.233,-50.782,-179.038,6.127,148.818
C07941=1179.038,90.482,-50.800,-179.035,6.129,148.817
C07942=1179.034,90.732,-50.818,-179.033,6.130,148.817
C07943=1179.029,90.981,-50.836,-179.030,6.131,148.816
C07944=1179.024,91.230,-50.854,-179.027,6.133,148.816
C07945=1179.019,91.480,-50.871,-179.025,6.134,148.815
C07946=1179.014,91.729,-50.889,-179.022,6.135,148.815
C07947=1179.009,91.978,-50.907,-179.019,6.136,148.814
C07948=1179.004,92.228,-50.925,-179.017,6.137,148.814
C07949=1178.999,92.477,-50.943,-179.014,6.138,148.813
C07950=1178.994,92.726,-50.961,-179.011,6.140,148.813
C07951=1178.990,92.976,-50.980,-179.009,6.140,148.812
C07952=1178.985,93.225,-50.998,-179.006,6.142,148.812
C07953=1178.980,93.474,-51.016,-179.004,6.143,148.811
C07954=1178.975,93.723,-51.034,-179.001,6.144,148.811
C07955=1178.970,93.973,-51.052,-178.998,6.145,148.810
C07956=1178.965,94.222,-51.070,-178.995,6.147,148.810
C07957=1178.960,94.471,-51.088,-178.993,6.147,148.809
C07958=1178.955,94.720,-51.106,-178.990,6.149,148.809
C07959=1178.951,94.970,-51.124,-178.988,6.150,148.808
C07960=1178.946,95.219,-51.142,-178.985,6.151,148.808
C07961=1178.941,95.469,-51.160,-178.982,6.153,148.807
C07962=1178.936,95.718,-51.178,-178.980,6.154,148.807
C07963=1178.931,95.967,-51.196,-178.977,6.155,148.806
C07964=1178.926,96.216,-51.214,-178.974,6.156,148.806
C07965=1178.922,96.466,-51.233,-178.972,6.158,148.805
C07966=1178.916,96.716,-51.251,-178.969,6.158,148.805
C07967=1178.911,96.965,-51.269,-178.966,6.160,148.804
C07968=1178.906,97.214,-51.287,-178.964,6.161,148.804
C07969=1178.902,97.462,-51.306,-178.961,6.162,148.803
C07970=1178.897,97.712,-51.324,-178.959,6.163,148.803
C07971=1178.893,97.961,-51.342,-178.956,6.165,148.802
C07972=1178.888,98.211,-51.360,-178.953,6.166,148.802
C07973=1178.882,98.460,-51.379,-178.951,6.167,148.801
C07974=1178.878,98.710,-51.397,-178.948,6.169,148.801
C07975=1178.873,98.959,-51.416,-178.945,6.169,148.800
C07976=1178.868,99.208,-51.434,-178.942,6.171,148.799
C07977=1178.863,99.457,-51.452,-178.940,6.172,148.799
C07978=1178.858,99.706,-51.470,-178.937,6.173,148.799
C07979=1178.853,99.956,-51.489,-178.934,6.175,148.798
C07980=1178.849,100.205,-51.507,-178.932,6.176,148.798
C07981=1178.844,100.454,-51.525,-178.929,6.177,148.797
C07982=1178.839,100.703,-51.543,-178.927,6.178,148.797
C07983=1178.834,100.953,-51.562,-178.924,6.180,148.796
C07984=1178.829,101.202,-51.581,-178.921,6.180,148.795
C07985=1178.824,101.451,-51.599,-178.919,6.182,148.795
C07986=1178.820,101.701,-51.617,-178.916,6.184,148.795
C07987=1178.815,101.950,-51.637,-178.913,6.184,148.794
C07988=1178.810,102.199,-51.655,-178.911,6.186,148.794
C07989=1178.805,102.448,-51.673,-178.908,6.187,148.793
C07990=1178.800,102.698,-51.691,-178.905,6.188,148.793
C07991=1178.795,102.947,-51.710,-178.903,6.190,148.792
C07992=1178.790,103.196,-51.728,-178.900,6.191,148.791
C07993=1178.786,103.446,-51.748,-178.897,6.192,148.791
C07994=1178.781,103.695,-51.766,-178.895,6.193,148.791
C07995=1178.776,103.944,-51.784,-178.892,6.195,148.790
C07996=1178.771,104.194,-51.803,-178.889,6.196,148.790
C07997=1178.766,104.443,-51.821,-178.887,6.197,148.789
C07998=1178.761,104.692,-51.839,-178.884,6.199,148.789
C07999=1178.756,104.942,-51.859,-178.882,6.199,148.788
C08000=1178.751,105.191,-51.877,-178.879,6.201,148.788
C08001=1178.747,105.439,-51.896,-178.876,6.203,148.787
C08002=1178.742,105.689,-51.915,-178.874,6.203,148.787
C08003=1178.737,105.938,-51.933,-178.871,6.205,148.786
C08004=1178.731,106.207,-51.953,-178.868,6.207,148.786
C08005=1178.727,106.476,-51.973,-178.865,6.207,148.785
C08006=1178.721,106.744,-51.994,-178.862,6.209,148.785
C08007=1178.716,107.012,-52.013,-178.859,6.210,148.784
C08008=1178.711,107.261,-52.033,-178.857,6.212,148.784
C08009=1178.707,107.511,-52.051,-178.854,6.213,148.783
C08010=1178.701,107.759,-52.070,-178.851,6.214,148.783
C08011=1178.697,108.009,-52.089,-178.849,6.216,148.782
C08012=1178.692,108.258,-52.107,-178.846,6.217,148.782
C08013=1178.687,108.507,-52.126,-178.843,6.218,148.781
C08014=1178.683,108.757,-52.145,-178.841,6.219,148.781
C08015=1178.677,109.005,-52.164,-178.838,6.221,148.780
C08016=1178.673,109.255,-52.183,-178.835,6.222,148.780
C08017=1178.668,109.504,-52.202,-178.833,6.223,148.779
C08018=1178.663,109.754,-52.220,-178.830,6.225,148.779
C08019=1178.658,110.003,-52.239,-178.827,6.226,148.778
C08020=1178.653,110.251,-52.258,-178.825,6.227,148.778
C08021=1178.648,110.502,-52.277,-178.822,6.229,148.777
C08022=1178.644,110.750,-52.296,-178.819,6.230,148.777
C08023=1178.639,111.000,-52.315,-178.817,6.231,148.776
C08024=1178.634,111.249,-52.333,-178.814,6.233,148.776
C08025=1178.629,111.499,-52.353,-178.812,6.233,148.775
C08026=1178.625,111.747,-52.372,-178.809,6.235,148.775
C08027=1178.619,111.997,-52.390,-178.806,6.237,148.774
C08028=1178.614,112.246,-52.410,-178.804,6.238,148.774
C08029=1178.610,112.495,-52.429,-178.801,6.239,148.773
C08030=1178.605,112.744,-52.448,-178.798,6.241,148.773
C08031=1178.600,112.993,-52.466,-178.796,6.242,148.773
C08032=1178.595,113.243,-52.486,-178.793,6.243,148.772
C08033=1178.591,113.492,-52.505,-178.790,6.245,148.772
C08034=1178.586,113.741,-52.524,-178.788,6.246,148.771
C08035=1178.580,113.991,-52.543,-178.785,6.247,148.771
C08036=1178.576,114.240,-52.562,-178.782,6.249,148.770
C08037=1178.571,114.489,-52.581,-178.780,6.250,148.770
C08038=1178.566,114.738,-52.601,-178.777,6.251,148.769
C08039=1178.562,114.987,-52.620,-178.774,6.253,148.769
C08040=1178.557,115.237,-52.639,-178.772,6.254,148.768
C08041=1178.552,115.486,-52.657,-178.769,6.255,148.768
C08042=1178.547,115.735,-52.677,-178.766,6.257,148.767
C08043=1178.542,115.984,-52.696,-178.764,6.258,148.767
C08044=1178.538,116.233,-52.715,-178.761,6.260,148.766
C08045=1178.533,116.482,-52.735,-178.758,6.261,148.766
C08046=1178.528,116.732,-52.754,-178.756,6.262,148.765
C08047=1178.524,116.981,-52.773,-178.753,6.264,148.765
C08048=1178.519,117.230,-52.793,-178.750,6.265,148.764
C08049=1178.513,117.480,-52.811,-178.748,6.266,148.764
C08050=1178.508,117.729,-52.831,-178.745,6.268,148.764
C08051=1178.504,117.978,-52.850,-178.743,6.270,148.763
C08052=1178.499,118.227,-52.869,-178.739,6.271,148.763
C08053=1178.494,118.477,-52.889,-178.737,6.272,148.762
C08054=1178.489,118.726,-52.908,-178.734,6.274,148.762
C08055=1178.485,118.975,-52.927,-178.731,6.275,148.761
C08056=1178.480,119.224,-52.947,-178.729,6.276,148.761
C08057=1178.475,119.473,-52.966,-178.726,6.278,148.760
C08058=1178.470,119.723,-52.986,-178.724,6.279,148.760
C08059=1178.466,119.972,-53.005,-178.721,6.280,148.759
C08060=1178.461,120.221,-53.024,-178.718,6.282,148.759
C08061=1178.456,120.470,-53.044,-178.716,6.283,148.758
C08062=1178.450,120.719,-53.063,-178.713,6.285,148.758
C08063=1178.447,120.968,-53.083,-178.710,6.286,148.757
C08064=1178.442,121.217,-53.102,-178.708,6.287,148.757
C08065=1178.437,121.466,-53.122,-178.705,6.289,148.757
C08066=1178.432,121.716,-53.141,-178.702,6.290,148.756
C08067=1178.427,121.965,-53.161,-178.700,6.291,148.756
C08068=1178.422,122.214,-53.180,-178.697,6.293,148.755
C08069=1178.418,122.464,-53.199,-178.694,6.295,148.755
C08070=1178.412,122.712,-53.219,-178.692,6.296,148.754
C08071=1178.408,122.962,-53.238,-178.689,6.297,148.754
C08072=1178.403,123.211,-53.259,-178.686,6.299,148.753
C08073=1178.398,123.460,-53.278,-178.684,6.301,148.753
C08074=1178.393,123.709,-53.298,-178.681,6.301,148.752
C08075=1178.388,123.959,-53.317,-178.678,6.303,148.752
C08076=1178.384,124.208,-53.336,-178.676,6.305,148.752
C08077=1178.379,124.457,-53.356,-178.673,6.306,148.751
C08078=1178.375,124.706,-53.376,-178.670,6.307,148.751
C08079=1178.370,124.956,-53.396,-178.668,6.309,148.750
C08080=1178.365,125.205,-53.415,-178.665,6.311,148.750
C08081=1178.360,125.453,-53.435,-178.663,6.312,148.749
C08082=1178.355,125.703,-53.455,-178.660,6.313,148.749
C08083=1178.350,125.952,-53.474,-178.657,6.315,148.748
C08084=1178.345,126.201,-53.494,-178.654,6.316,148.748
C08085=1178.341,126.450,-53.514,-178.652,6.317,148.747
C08086=1178.336,126.700,-53.534,-178.649,6.319,148.747
C08087=1178.331,126.949,-53.553,-178.646,6.320,148.746
C08088=1178.326,127.198,-53.574,-178.643,6.322,148.746
C08089=1178.322,127.447,-53.593,-178.641,6.323,148.746
C08090=1178.317,127.697,-53.613,-178.639,6.325,148.745
C08091=1178.312,127.945,-53.633,-178.635,6.326,148.745
C08092=1178.307,128.195,-53.653,-178.633,6.328,148.744
C08093=1178.303,128.444,-53.673,-178.631,6.329,148.744
C08094=1178.298,128.693,-53.693,-178.628,6.331,148.743
C08095=1178.293,128.942,-53.712,-178.625,6.332,148.743
C08096=1178.288,129.191,-53.732,-178.622,6.334,148.742
C08097=1178.283,129.441,-53.752,-178.620,6.335,148.742
C08098=1178.279,129.690,-53.772,-178.617,6.336,148.742
C08099=1178.274,129.938,-53.792,-178.614,6.338,148.741
C08100=1178.269,130.187,-53.812,-178.611,6.340,148.741
C08101=1178.264,130.437,-53.832,-178.609,6.341,148.740
C08102=1178.260,130.687,-53.851,-178.606,6.342,148.740
C08103=1178.255,130.936,-53.872,-178.604,6.344,148.739
C08104=1178.250,131.184,-53.891,-178.601,6.346,148.739
C08105=1178.245,131.433,-53.911,-178.598,6.347,148.738
C08106=1178.240,131.683,-53.932,-178.596,6.348,148.738
C08107=1178.236,131.932,-53.952,-178.593,6.350,148.738
C08108=1178.231,132.201,-53.973,-178.590,6.352,148.737
C08109=1178.225,132.469,-53.995,-178.587,6.353,148.737
C08110=1178.220,132.738,-54.017,-178.584,6.355,148.736
C08111=1178.215,133.007,-54.038,-178.581,6.356,148.736
C08112=1178.210,133.256,-54.059,-178.579,6.358,148.735
C08113=1178.206,133.505,-54.079,-178.576,6.360,148.735
C08114=1178.201,133.754,-54.099,-178.573,6.361,148.734
C08115=1178.196,134.002,-54.119,-178.571,6.363,148.734
C08116=1178.192,134.251,-54.139,-178.568,6.364,148.733
C08117=1178.186,134.501,-54.159,-178.565,6.365,148.733
C08118=1178.182,134.750,-54.180,-178.563,6.367,148.733
C08119=1178.177,135.000,-54.199,-178.560,6.369,148.732
C08120=1178.173,135.249,-54.220,-178.557,6.371,148.732
C08121=1178.168,135.498,-54.240,-178.555,6.372,148.732
C08122=1178.163,135.747,-54.261,-178.552,6.373,148.731
C08123=1178.158,135.996,-54.280,-178.549,6.375,148.731
C08124=1178.153,136.245,-54.301,-178.546,6.376,148.730
C08125=1178.149,136.494,-54.321,-178.544,6.378,148.730
C08126=1178.143,136.744,-54.341,-178.542,6.379,148.729
C08127=1178.139,136.993,-54.362,-178.539,6.381,148.729
C08128=1178.134,137.242,-54.382,-178.536,6.382,148.728
C08129=1178.130,137.490,-54.402,-178.533,6.384,148.728
C08130=1178.124,137.740,-54.423,-178.530,6.386,148.728
C08131=1178.120,137.989,-54.443,-178.528,6.388,148.727
C08132=1178.116,138.238,-54.463,-178.526,6.388,148.727
C08133=1178.110,138.487,-54.484,-178.523,6.390,148.726
C08134=1178.106,138.736,-54.505,-178.520,6.392,148.726
C08135=1178.101,138.986,-54.524,-178.517,6.393,148.725
C08136=1178.096,139.235,-54.545,-178.514,6.395,148.725
C08137=1178.091,139.484,-54.565,-178.512,6.397,148.725
C08138=1178.087,139.732,-54.586,-178.509,6.398,148.724
C08139=1178.081,139.982,-54.607,-178.507,6.400,148.724
C08140=1178.077,140.231,-54.627,-178.504,6.401,148.723
C08141=1178.073,140.480,-54.647,-178.501,6.403,148.723
C08142=1178.067,140.729,-54.668,-178.498,6.404,148.722
C08143=1178.063,140.978,-54.688,-178.495,6.406,148.722
C08144=1178.058,141.227,-54.708,-178.493,6.407,148.722
C08145=1178.053,141.477,-54.729,-178.491,6.409,148.721
C08146=1178.049,141.726,-54.750,-178.488,6.411,148.721
C08147=1178.043,141.975,-54.771,-178.485,6.412,148.720
C08148=1178.039,142.224,-54.791,-178.482,6.414,148.720
C08149=1178.034,142.473,-54.812,-178.479,6.416,148.720
C08150=1178.029,142.722,-54.832,-178.477,6.417,148.719
C08151=1178.025,142.971,-54.853,-178.475,6.418,148.719
C08152=1178.020,143.221,-54.874,-178.472,6.420,148.718
C08153=1178.016,143.470,-54.895,-178.469,6.422,148.718
C08154=1178.011,143.719,-54.916,-178.466,6.423,148.717
C08155=1178.006,143.968,-54.936,-178.463,6.425,148.717
C08156=1178.002,144.217,-54.956,-178.461,6.427,148.717
C08157=1177.997,144.466,-54.977,-178.458,6.428,148.716
C08158=1177.993,144.715,-54.998,-178.455,6.430,148.716
C08159=1177.987,144.964,-55.019,-178.453,6.431,148.715
C08160=1177.983,145.213,-55.040,-178.450,6.433,148.715
C08161=1177.978,145.462,-55.061,-178.448,6.435,148.715
C08162=1177.973,145.711,-55.081,-178.445,6.436,148.714
C08163=1177.968,145.960,-55.102,-178.442,6.438,148.714
C08164=1177.964,146.209,-55.122,-178.439,6.439,148.713
C08165=1177.958,146.459,-55.143,-178.436,6.441,148.713
C08166=1177.955,146.708,-55.165,-178.434,6.443,148.713
C08167=1177.950,146.957,-55.186,-178.432,6.444,148.712
C08168=1177.945,147.206,-55.207,-178.429,6.446,148.712
C08169=1177.940,147.455,-55.227,-178.426,6.447,148.711
C08170=1177.935,147.704,-55.248,-178.424,6.449,148.711
C08171=1177.931,147.953,-55.268,-178.421,6.451,148.711
C08172=1177.926,148.202,-55.290,-178.418,6.452,148.710
C08173=1177.921,148.451,-55.310,-178.415,6.454,148.710
C08174=1177.916,148.700,-55.331,-178.412,6.456,148.709
C08175=1177.912,148.950,-55.353,-178.410,6.458,148.709
C08176=1177.907,149.198,-55.374,-178.407,6.459,148.708
C08177=1177.902,149.448,-55.395,-178.405,6.460,148.708
C08178=1177.897,149.697,-55.416,-178.402,6.462,148.708
C08179=1177.893,149.945,-55.437,-178.399,6.464,148.707
C08180=1177.888,150.194,-55.458,-178.397,6.466,148.707
C08181=1177.883,150.444,-55.479,-178.394,6.467,148.707
C08182=1177.879,150.693,-55.500,-178.391,6.469,148.706
C08183=1177.874,150.942,-55.521,-178.388,6.471,148.706
C08184=1177.869,151.191,-55.542,-178.386,6.472,148.705
C08185=1177.865,151.440,-55.563,-178.383,6.474,148.705
C08186=1177.859,151.689,-55.584,-178.380,6.476,148.704
C08187=1177.855,151.939,-55.606,-178.377,6.478,148.704
C08188=1177.851,152.187,-55.627,-178.375,6.479,148.704
C08189=1177.845,152.436,-55.648,-178.373,6.480,148.703
C08190=1177.841,152.685,-55.669,-178.370,6.482,148.703
C08191=1177.836,152.934,-55.690,-178.367,6.484,148.703
C08192=1177.832,153.184,-55.711,-178.365,6.486,148.702
C08193=1177.827,153.433,-55.733,-178.362,6.487,148.702
C08194=1177.822,153.682,-55.754,-178.359,6.489,148.701
C08195=1177.817,153.930,-55.775,-178.357,6.491,148.701
C08196=1177.812,154.179,-55.796,-178.354,6.493,148.701
C08197=1177.808,154.429,-55.818,-178.351,6.494,148.700
C08198=1177.803,154.678,-55.839,-178.348,6.496,148.700
C08199=1177.798,154.927,-55.860,-178.345,6.497,148.699
C08200=1177.794,155.176,-55.881,-178.343,6.499,148.699
C08201=1177.789,155.425,-55.903,-178.340,6.501,148.699
C08202=1177.784,155.674,-55.925,-178.337,6.503,148.698
C08203=1177.779,155.923,-55.945,-178.335,6.505,148.698
C08204=1177.775,156.172,-55.968,-178.332,6.506,148.697
C08205=1177.770,156.421,-55.988,-178.329,6.508,148.697
C08206=1177.766,156.670,-56.010,-178.327,6.509,148.697
C08207=1177.760,156.919,-56.031,-178.324,6.511,148.696
C08208=1177.756,157.168,-56.053,-178.322,6.513,148.696
C08209=1177.751,157.417,-56.074,-178.319,6.514,148.696
C08210=1177.746,157.666,-56.095,-178.316,6.516,148.695
C08211=1177.742,157.916,-56.117,-178.314,6.518,148.695
C08212=1177.737,158.185,-56.140,-178.311,6.520,148.694
C08213=1177.731,158.453,-56.163,-178.308,6.522,148.694
C08214=1177.727,158.722,-56.187,-178.304,6.524,148.693
C08215=1177.721,158.991,-56.210,-178.302,6.525,148.693
C08216=1177.718,159.240,-56.231,-178.299,6.527,148.693
C08217=1177.713,159.489,-56.253,-178.296,6.529,148.692
C08218=1177.708,159.738,-56.274,-178.294,6.531,148.692
C08219=1177.703,159.987,-56.296,-178.291,6.532,148.692
C08220=1177.698,160.236,-56.318,-178.288,6.534,148.691
C08221=1177.694,160.485,-56.339,-178.286,6.536,148.691
C08222=1177.689,160.735,-56.361,-178.283,6.538,148.690
C08223=1177.684,160.983,-56.382,-178.280,6.539,148.690
C08224=1177.679,161.232,-56.404,-178.278,6.541,148.690
C08225=1177.675,161.481,-56.426,-178.275,6.543,148.689
C08226=1177.670,161.731,-56.447,-178.272,6.545,148.689
C08227=1177.666,161.980,-56.469,-178.270,6.546,148.689
C08228=1177.661,162.229,-56.491,-178.267,6.548,148.688
C08229=1177.656,162.477,-56.513,-178.264,6.550,148.688
C08230=1177.651,162.727,-56.535,-178.262,6.552,148.687
C08231=1177.647,162.975,-56.556,-178.259,6.554,148.687
C08232=1177.642,163.224,-56.578,-178.256,6.555,148.687
C08233=1177.637,163.473,-56.600,-178.253,6.557,148.686
C08234=1177.632,163.722,-56.621,-178.251,6.559,148.686
C08235=1177.628,163.972,-56.643,-178.248,6.561,148.686
C08236=1177.623,164.220,-56.665,-178.245,6.562,148.685
C08237=1177.619,164.470,-56.687,-178.243,6.564,148.685
C08238=1177.614,164.718,-56.708,-178.240,6.566,148.685
C08239=1177.610,164.968,-56.730,-178.237,6.568,148.684
C08240=1177.604,165.217,-56.753,-178.235,6.569,148.684
C08241=1177.600,165.466,-56.775,-178.232,6.571,148.683
C08242=1177.595,165.715,-56.796,-178.229,6.573,148.683
C08243=1177.590,165.963,-56.818,-178.227,6.575,148.683
C08244=1177.586,166.213,-56.840,-178.224,6.576,148.682
C08245=1177.581,166.461,-56.862,-178.221,6.578,148.682
C08246=1177.577,166.711,-56.884,-178.219,6.580,148.682
C08247=1177.572,166.959,-56.906,-178.216,6.582,148.681
C08248=1177.567,167.209,-56.928,-178.213,6.584,148.681
C08249=1177.562,167.458,-56.950,-178.211,6.585,148.680
C08250=1177.558,167.707,-56.972,-178.208,6.587,148.680
C08251=1177.553,167.955,-56.994,-178.205,6.589,148.680
C08252=1177.549,168.204,-57.016,-178.202,6.591,148.679
C08253=1177.544,168.453,-57.038,-178.200,6.592,148.679
C08254=1177.539,168.703,-57.061,-178.197,6.594,148.679
C08255=1177.534,168.951,-57.082,-178.195,6.596,148.678
C08256=1177.530,169.201,-57.104,-178.192,6.599,148.678
C08257=1177.525,169.449,-57.126,-178.189,6.601,148.678
C08258=1177.520,169.698,-57.150,-178.186,6.602,148.677
C08259=1177.515,169.947,-57.171,-178.184,6.604,148.677
C08260=1177.511,170.196,-57.193,-178.181,6.606,148.677
C08261=1177.507,170.446,-57.215,-178.178,6.608,148.676
C08262=1177.501,170.694,-57.238,-178.176,6.609,148.676
C08263=1177.497,170.943,-57.260,-178.173,6.611,148.676
C08264=1177.492,171.192,-57.282,-178.170,6.613,148.675
C08265=1177.488,171.441,-57.304,-178.168,6.615,148.675
C08266=1177.483,171.690,-57.326,-178.165,6.617,148.674
C08267=1177.479,171.939,-57.349,-178.162,6.618,148.674
C08268=1177.474,172.187,-57.371,-178.159,6.620,148.674
C08269=1177.469,172.437,-57.393,-178.157,6.622,148.673
C08270=1177.465,172.686,-57.416,-178.154,6.624,148.673
C08271=1177.460,172.934,-57.438,-178.151,6.625,148.673
C08272=1177.455,173.184,-57.461,-178.149,6.628,148.672
C08273=1177.450,173.432,-57.483,-178.146,6.630,148.672
C08274=1177.446,173.681,-57.505,-178.143,6.632,148.672
C08275=1177.441,173.931,-57.528,-178.141,6.634,148.671
C08276=1177.437,174.179,-57.550,-178.138,6.635,148.671
C08277=1177.432,174.429,-57.572,-178.135,6.637,148.671
C08278=1177.427,174.677,-57.594,-178.133,6.639,148.670
C08279=1177.423,174.926,-57.617,-178.130,6.641,148.670
C08280=1177.418,175.176,-57.639,-178.127,6.643,148.670
C08281=1177.413,175.424,-57.662,-178.125,6.644,148.669
C08282=1177.409,175.673,-57.684,-178.122,6.646,148.669
C08283=1177.404,175.922,-57.708,-178.119,6.648,148.669
C08284=1177.399,176.171,-57.729,-178.117,6.650,148.668
C08285=1177.394,176.421,-57.752,-178.114,6.653,148.668
C08286=1177.390,176.669,-57.775,-178.111,6.654,148.668
C08287=1177.385,176.918,-57.796,-178.108,6.656,148.667
C08288=1177.381,177.167,-57.820,-178.106,6.658,148.667
C08289=1177.377,177.416,-57.842,-178.103,6.660,148.667
C08290=1177.371,177.665,-57.865,-178.100,6.661,148.666
C08291=1177.367,177.913,-57.888,-178.098,6.663,148.666
C08292=1177.362,178.163,-57.910,-178.095,6.665,148.665
C08293=1177.358,178.411,-57.933,-178.092,6.667,148.665
C08294=1177.353,178.661,-57.955,-178.090,6.669,148.665
C08295=1177.349,178.909,-57.978,-178.087,6.671,148.665
C08296=1177.344,179.158,-58.001,-178.084,6.673,148.664
C08297=1177.339,179.407,-58.023,-178.082,6.675,148.664
C08298=1177.334,179.656,-58.046,-178.079,6.677,148.664
C08299=1177.330,179.905,-58.068,-178.076,6.679,148.663
C08300=1177.325,180.154,-58.092,-178.073,6.680,148.663
C08301=1177.321,180.402,-58.114,-178.071,6.682,148.662
C08302=1177.316,180.652,-58.137,-178.069,6.684,148.662
C08303=1177.311,180.901,-58.160,-178.065,6.687,148.662
C08304=1177.307,181.150,-58.183,-178.063,6.689,148.662
C08305=1177.302,181.399,-58.205,-178.060,6.690,148.661
C08306=1177.298,181.648,-58.228,-178.057,6.692,148.661
C08307=1177.293,181.897,-58.251,-178.055,6.694,148.661
C08308=1177.289,182.145,-58.274,-178.052,6.696,148.660
C08309=1177.283,182.394,-58.296,-178.050,6.698,148.660
C08310=1177.279,182.643,-58.320,-178.047,6.700,148.660
C08311=1177.275,182.892,-58.342,-178.044,6.702,148.659
C08312=1177.270,183.141,-58.366,-178.041,6.704,148.659
C08313=1177.265,183.390,-58.389,-178.038,6.706,148.659
C08314=1177.260,183.639,-58.411,-178.036,6.708,148.658
C08315=1177.256,183.888,-58.434,-178.033,6.709,148.658
C08316=1177.250,184.157,-58.459,-178.030,6.712,148.658
C08317=1177.246,184.427,-58.484,-178.027,6.714,148.657
C08318=1177.241,184.697,-58.509,-178.025,6.715,148.657
C08319=1177.236,184.966,-58.534,-178.021,6.718,148.657
C08320=1177.231,185.215,-58.557,-178.019,6.720,148.656
C08321=1177.227,185.464,-58.580,-178.016,6.722,148.656
C08322=1177.222,185.713,-58.603,-178.014,6.724,148.656
C08323=1177.218,185.962,-58.626,-178.011,6.726,148.655
C08324=1177.213,186.210,-58.649,-178.008,6.728,148.655
C08325=1177.208,186.459,-58.672,-178.005,6.730,148.655
C08326=1177.204,186.708,-58.695,-178.003,6.732,148.655
C08327=1177.199,186.957,-58.719,-178.000,6.734,148.654
C08328=1177.195,187.206,-58.742,-177.998,6.736,148.654
C08329=1177.190,187.455,-58.765,-177.994,6.738,148.654
C08330=1177.185,187.704,-58.789,-177.992,6.740,148.653
C08331=1177.181,187.952,-58.811,-177.990,6.742,148.653
C08332=1177.176,188.201,-58.834,-177.987,6.744,148.653
C08333=1177.171,188.450,-58.858,-177.984,6.746,148.652
C08334=1177.166,188.699,-58.881,-177.981,6.747,148.652
C08335=1177.162,188.948,-58.904,-177.978,6.750,148.652
C08336=1177.158,189.197,-58.927,-177.976,6.752,148.651
C08337=1177.153,189.446,-58.951,-177.973,6.754,148.651
C08338=1177.148,189.695,-58.974,-177.971,6.756,148.651
C08339=1177.144,189.944,-58.997,-177.968,6.757,148.650
C08340=1177.139,190.193,-59.021,-177.965,6.760,148.650
C08341=1177.135,190.442,-59.045,-177.962,6.762,148.650
C08342=1177.129,190.690,-59.068,-177.960,6.764,148.650
C08343=1177.125,190.939,-59.090,-177.957,6.766,148.649
C08344=1177.121,191.188,-59.114,-177.955,6.768,148.649
C08345=1177.116,191.437,-59.137,-177.951,6.770,148.649
C08346=1177.111,191.686,-59.161,-177.949,6.772,148.648
C08347=1177.107,191.934,-59.185,-177.946,6.774,148.648
C08348=1177.102,192.183,-59.208,-177.944,6.776,148.648
C08349=1177.097,192.432,-59.231,-177.941,6.778,148.647
C08350=1177.093,192.681,-59.255,-177.938,6.780,148.647
C08351=1177.088,192.930,-59.278,-177.936,6.782,148.647
C08352=1177.084,193.179,-59.302,-177.933,6.784,148.647
C08353=1177.079,193.428,-59.325,-177.930,6.786,148.646
C08354=1177.074,193.677,-59.349,-177.928,6.788,148.646
C08355=1177.070,193.926,-59.372,-177.924,6.790,148.646
C08356=1177.065,194.174,-59.396,-177.922,6.792,148.645
C08357=1177.060,194.423,-59.420,-177.920,6.794,148.645
C08358=1177.056,194.672,-59.443,-177.917,6.796,148.645
C08359=1177.051,194.921,-59.467,-177.914,6.798,148.644
C08360=1177.047,195.170,-59.490,-177.911,6.801,148.644
C08361=1177.042,195.419,-59.514,-177.909,6.803,148.644
C08362=1177.038,195.667,-59.538,-177.906,6.804,148.644
C08363=1177.033,195.916,-59.561,-177.903,6.806,148.643
C08364=1177.028,196.165,-59.585,-177.901,6.809,148.643
C08365=1177.024,196.414,-59.609,-177.898,6.811,148.643
C08366=1177.019,196.663,-59.632,-177.895,6.813,148.642
C08367=1177.015,196.911,-59.656,-177.893,6.814,148.642
C08368=1177.010,197.160,-59.679,-177.890,6.817,148.642
C08369=1177.006,197.409,-59.704,-177.887,6.819,148.642
C08370=1177.002,197.658,-59.727,-177.885,6.821,148.641
C08371=1176.997,197.907,-59.751,-177.882,6.823,148.641
C08372=1176.992,198.156,-59.775,-177.879,6.826,148.641
C08373=1176.988,198.404,-59.799,-177.876,6.827,148.640
C08374=1176.983,198.653,-59.823,-177.874,6.829,148.640
C08375=1176.978,198.902,-59.847,-177.871,6.831,148.640
C08376=1176.973,199.151,-59.870,-177.868,6.834,148.640
C08377=1176.969,199.399,-59.894,-177.866,6.836,148.639
C08378=1176.964,199.648,-59.918,-177.863,6.838,148.639
C08379=1176.961,199.897,-59.942,-177.861,6.840,148.639
C08380=1176.956,200.147,-59.965,-177.858,6.842,148.639
C08381=1176.951,200.395,-59.990,-177.855,6.844,148.638
C08382=1176.946,200.644,-60.014,-177.852,6.846,148.638
C08383=1176.942,200.893,-60.037,-177.850,6.848,148.638
C08384=1176.937,201.141,-60.062,-177.847,6.851,148.637
C08385=1176.933,201.390,-60.085,-177.844,6.852,148.637
C08386=1176.927,201.639,-60.110,-177.842,6.855,148.637
C08387=1176.924,201.888,-60.134,-177.839,6.857,148.637
C08388=1176.919,202.137,-60.157,-177.836,6.859,148.636
C08389=1176.915,202.385,-60.181,-177.833,6.861,148.636
C08390=1176.910,202.634,-60.206,-177.831,6.863,148.636
C08391=1176.905,202.883,-60.229,-177.828,6.865,148.635
C08392=1176.901,203.132,-60.254,-177.825,6.867,148.635
C08393=1176.897,203.381,-60.278,-177.823,6.869,148.635
C08394=1176.892,203.629,-60.302,-177.820,6.871,148.635
C08395=1176.887,203.878,-60.326,-177.817,6.874,148.634
C08396=1176.882,204.127,-60.350,-177.815,6.876,148.634
C08397=1176.879,204.376,-60.375,-177.812,6.878,148.634
C08398=1176.873,204.625,-60.399,-177.809,6.880,148.634
C08399=1176.869,204.873,-60.423,-177.806,6.882,148.633
C08400=1176.864,205.122,-60.447,-177.804,6.884,148.633
C08401=1176.859,205.371,-60.471,-177.801,6.887,148.633
C08402=1176.855,205.620,-60.496,-177.798,6.889,148.632
C08403=1176.851,205.868,-60.520,-177.796,6.891,148.632
C08404=1176.846,206.117,-60.544,-177.794,6.893,148.632
C08405=1176.841,206.366,-60.569,-177.790,6.895,148.632
C08406=1176.837,206.615,-60.592,-177.788,6.897,148.632
C08407=1176.832,206.864,-60.617,-177.785,6.899,148.631
C08408=1176.828,207.112,-60.641,-177.782,6.902,148.631
C08409=1176.823,207.361,-60.666,-177.780,6.904,148.631
C08410=1176.819,207.610,-60.690,-177.777,6.906,148.630
C08411=1176.815,207.859,-60.714,-177.774,6.908,148.630
C08412=1176.809,208.107,-60.739,-177.772,6.910,148.630
C08413=1176.805,208.356,-60.763,-177.769,6.912,148.630
C08414=1176.800,208.605,-60.788,-177.766,6.915,148.629
C08415=1176.796,208.854,-60.812,-177.764,6.917,148.629
C08416=1176.791,209.102,-60.837,-177.761,6.919,148.629
C08417=1176.787,209.351,-60.861,-177.758,6.921,148.629
C08418=1176.782,209.600,-60.886,-177.756,6.923,148.628
C08419=1176.778,209.849,-60.910,-177.753,6.925,148.628
C08420=1176.772,210.119,-60.937,-177.750,6.928,148.628
C08421=1176.768,210.390,-60.964,-177.748,6.930,148.628
C08422=1176.762,210.660,-60.990,-177.744,6.933,148.627
C08423=1176.757,210.931,-61.016,-177.741,6.935,148.627
C08424=1176.754,211.180,-61.041,-177.739,6.937,148.627
C08425=1176.749,211.428,-61.066,-177.736,6.939,148.627
C08426=1176.744,211.676,-61.090,-177.733,6.942,148.626
C08427=1176.740,211.926,-61.115,-177.730,6.944,148.626
C08428=1176.735,212.174,-61.139,-177.728,6.946,148.626
C08429=1176.731,212.423,-61.164,-177.725,6.948,148.625
C08430=1176.726,212.672,-61.189,-177.723,6.950,148.625
C08431=1176.721,212.921,-61.213,-177.720,6.952,148.625
C08432=1176.717,213.169,-61.239,-177.717,6.955,148.625
C08433=1176.713,213.418,-61.263,-177.715,6.957,148.625
C08434=1176.708,213.667,-61.288,-177.712,6.960,148.624
C08435=1176.704,213.916,-61.312,-177.709,6.961,148.624
C08436=1176.699,214.164,-61.338,-177.707,6.963,148.624
C08437=1176.694,214.413,-61.363,-177.703,6.966,148.624
C08438=1176.690,214.662,-61.387,-177.701,6.968,148.623
C08439=1176.685,214.910,-61.411,-177.699,6.970,148.623
C08440=1176.681,215.159,-61.436,-177.695,6.973,148.623
C08441=1176.676,215.408,-61.461,-177.693,6.975,148.623
C08442=1176.672,215.657,-61.486,-177.691,6.977,148.622
C08443=1176.668,215.905,-61.511,-177.688,6.980,148.622
C08444=1176.663,216.154,-61.536,-177.685,6.981,148.622
C08445=1176.658,216.403,-61.561,-177.682,6.984,148.622
C08446=1176.654,216.651,-61.585,-177.680,6.986,148.621
C08447=1176.649,216.900,-61.610,-177.677,6.988,148.621
C08448=1176.644,217.149,-61.635,-177.674,6.991,148.621
C08449=1176.640,217.398,-61.661,-177.672,6.993,148.621
C08450=1176.636,217.646,-61.685,-177.669,6.994,148.620
C08451=1176.631,217.895,-61.711,-177.666,6.997,148.620
C08452=1176.626,218.144,-61.735,-177.664,6.999,148.620
C08453=1176.623,218.392,-61.761,-177.661,7.002,148.620
C08454=1176.618,218.641,-61.785,-177.658,7.004,148.620
C08455=1176.613,218.890,-61.810,-177.656,7.006,148.619
C08456=1176.608,219.138,-61.836,-177.653,7.009,148.619
C08457=1176.604,219.388,-61.861,-177.650,7.010,148.619
C08458=1176.600,219.636,-61.885,-177.647,7.013,148.619
C08459=1176.595,219.885,-61.911,-177.645,7.015,148.618
C08460=1176.590,220.133,-61.936,-177.642,7.017,148.618
C08461=1176.586,220.382,-61.962,-177.639,7.020,148.618
C08462=1176.582,220.630,-61.986,-177.637,7.022,148.618
C08463=1176.577,220.879,-62.011,-177.634,7.025,148.618
C08464=1176.572,221.128,-62.036,-177.632,7.027,148.617
C08465=1176.568,221.377,-62.062,-177.629,7.029,148.617
C08466=1176.564,221.626,-62.087,-177.626,7.031,148.617
C08467=1176.559,221.874,-62.112,-177.624,7.033,148.617
C08468=1176.555,222.123,-62.138,-177.620,7.036,148.616
C08469=1176.550,222.371,-62.162,-177.618,7.038,148.616
C08470=1176.546,222.620,-62.188,-177.615,7.041,148.616
C08471=1176.541,222.868,-62.213,-177.613,7.043,148.616
C08472=1176.537,223.118,-62.238,-177.610,7.045,148.615
C08473=1176.532,223.367,-62.264,-177.607,7.048,148.615
C08474=1176.527,223.615,-62.289,-177.605,7.050,148.615
C08475=1176.523,223.864,-62.314,-177.602,7.052,148.615
C08476=1176.518,224.112,-62.340,-177.599,7.054,148.615
C08477=1176.514,224.361,-62.366,-177.596,7.057,148.615
C08478=1176.509,224.609,-62.391,-177.594,7.059,148.614
C08479=1176.505,224.858,-62.416,-177.592,7.061,148.614
C08480=1176.500,225.107,-62.442,-177.588,7.064,148.614
C08481=1176.496,225.355,-62.467,-177.586,7.066,148.614
C08482=1176.492,225.604,-62.492,-177.583,7.069,148.613
C08483=1176.488,225.853,-62.518,-177.580,7.070,148.613
C08484=1176.483,226.101,-62.543,-177.578,7.073,148.613
C08485=1176.478,226.350,-62.568,-177.575,7.075,148.613
C08486=1176.474,226.599,-62.594,-177.572,7.078,148.613
C08487=1176.469,226.847,-62.620,-177.570,7.080,148.612
C08488=1176.464,227.096,-62.646,-177.567,7.082,148.612
C08489=1176.460,227.344,-62.671,-177.564,7.085,148.612
C08490=1176.455,227.593,-62.697,-177.562,7.087,148.612
C08491=1176.451,227.843,-62.722,-177.559,7.089,148.611
C08492=1176.446,228.091,-62.748,-177.557,7.092,148.611
C08493=1176.442,228.339,-62.773,-177.554,7.094,148.611
C08494=1176.438,228.588,-62.799,-177.551,7.096,148.611
C08495=1176.433,228.837,-62.825,-177.548,7.099,148.611
C08496=1176.429,229.085,-62.850,-177.546,7.101,148.611
C08497=1176.424,229.334,-62.876,-177.543,7.104,148.610
C08498=1176.420,229.583,-62.902,-177.540,7.106,148.610
C08499=1176.415,229.831,-62.927,-177.538,7.108,148.610
C08500=1176.411,230.080,-62.953,-177.535,7.111,148.610
C08501=1176.406,230.329,-62.979,-177.533,7.113,148.610
C08502=1176.402,230.578,-63.005,-177.529,7.115,148.609
C08503=1176.397,230.826,-63.030,-177.527,7.117,148.609
C08504=1176.393,231.075,-63.056,-177.524,7.120,148.609
C08505=1176.389,231.323,-63.082,-177.522,7.122,148.609
C08506=1176.384,231.571,-63.107,-177.519,7.125,148.609
C08507=1176.379,231.820,-63.134,-177.517,7.127,148.608
C08508=1176.375,232.069,-63.160,-177.514,7.130,148.608
C08509=1176.371,232.318,-63.186,-177.511,7.132,148.608
C08510=1176.366,232.566,-63.211,-177.508,7.135,148.608
C08511=1176.362,232.814,-63.237,-177.506,7.137,148.608
C08512=1176.357,233.064,-63.263,-177.503,7.140,148.608
C08513=1176.352,233.312,-63.289,-177.500,7.141,148.607
C08514=1176.348,233.561,-63.315,-177.498,7.144,148.607
C08515=1176.344,233.809,-63.341,-177.495,7.146,148.607
C08516=1176.339,234.058,-63.367,-177.492,7.149,148.607
C08517=1176.334,234.307,-63.393,-177.490,7.151,148.607
C08518=1176.331,234.555,-63.419,-177.487,7.154,148.606
C08519=1176.326,234.804,-63.445,-177.485,7.156,148.606
C08520=1176.321,235.052,-63.471,-177.481,7.159,148.606
C08521=1176.317,235.301,-63.497,-177.479,7.161,148.606
C08522=1176.313,235.549,-63.523,-177.476,7.164,148.606
C08523=1176.308,235.798,-63.549,-177.474,7.166,148.605
C08524=1176.303,236.070,-63.578,-177.471,7.168,148.605
C08525=1176.299,236.341,-63.606,-177.468,7.171,148.605
C08526=1176.293,236.612,-63.634,-177.465,7.174,148.605
C08527=1176.288,236.884,-63.664,-177.462,7.177,148.605
C08528=1176.284,237.133,-63.689,-177.460,7.179,148.605
C08529=1176.279,237.381,-63.716,-177.456,7.181,148.604
C08530=1176.275,237.630,-63.742,-177.454,7.184,148.604
C08531=1176.271,237.879,-63.768,-177.451,7.187,148.604
C08532=1176.266,238.127,-63.795,-177.449,7.188,148.604
C08533=1176.262,238.376,-63.821,-177.446,7.191,148.604
C08534=1176.257,238.624,-63.847,-177.443,7.193,148.603
C08535=1176.252,238.873,-63.873,-177.441,7.196,148.603
C08536=1176.249,239.121,-63.900,-177.438,7.199,148.603
C08537=1176.244,239.370,-63.926,-177.435,7.201,148.603
C08538=1176.240,239.618,-63.952,-177.433,7.204,148.603
C08539=1176.235,239.867,-63.979,-177.430,7.206,148.603
C08540=1176.231,240.116,-64.005,-177.427,7.209,148.603
C08541=1176.227,240.364,-64.031,-177.425,7.211,148.602
C08542=1176.222,240.613,-64.058,-177.422,7.213,148.602
C08543=1176.218,240.862,-64.084,-177.420,7.216,148.602
C08544=1176.213,241.110,-64.111,-177.417,7.219,148.602
C08545=1176.209,241.359,-64.137,-177.414,7.220,148.602
C08546=1176.204,241.607,-64.163,-177.411,7.223,148.602
C08547=1176.200,241.855,-64.190,-177.409,7.226,148.601
C08548=1176.195,242.104,-64.216,-177.406,7.228,148.601
C08549=1176.191,242.352,-64.243,-177.403,7.231,148.601
C08550=1176.186,242.601,-64.269,-177.401,7.233,148.601
C08551=1176.181,242.850,-64.296,-177.398,7.236,148.601
C08552=1176.177,243.098,-64.322,-177.396,7.238,148.601
C08553=1176.172,243.347,-64.349,-177.393,7.241,148.601
C08554=1176.168,243.595,-64.375,-177.390,7.244,148.600
C08555=1176.164,243.844,-64.402,-177.388,7.246,148.600
C08556=1176.159,244.093,-64.428,-177.385,7.249,148.600
C08557=1176.155,244.341,-64.455,-177.382,7.250,148.600
C08558=1176.151,244.589,-64.482,-177.379,7.253,148.600
C08559=1176.146,244.838,-64.509,-177.377,7.256,148.600
C08560=1176.141,245.087,-64.535,-177.374,7.259,148.600
C08561=1176.137,245.335,-64.561,-177.371,7.261,148.599
C08562=1176.133,245.584,-64.588,-177.369,7.263,148.599
C08563=1176.128,245.832,-64.616,-177.366,7.266,148.599
C08564=1176.124,246.080,-64.642,-177.364,7.268,148.599
C08565=1176.119,246.330,-64.668,-177.361,7.271,148.599
C08566=1176.115,246.579,-64.696,-177.358,7.274,148.599
C08567=1176.111,246.827,-64.722,-177.356,7.276,148.598
C08568=1176.106,247.075,-64.749,-177.353,7.279,148.598
C08569=1176.102,247.324,-64.776,-177.351,7.281,148.598
C08570=1176.098,247.572,-64.803,-177.348,7.284,148.598
C08571=1176.093,247.821,-64.830,-177.345,7.286,148.598
C08572=1176.089,248.069,-64.857,-177.342,7.289,148.598
C08573=1176.085,248.317,-64.883,-177.340,7.292,148.598
C08574=1176.080,248.566,-64.910,-177.338,7.294,148.598
C08575=1176.075,248.815,-64.937,-177.334,7.296,148.597
C08576=1176.070,249.063,-64.964,-177.332,7.299,148.597
C08577=1176.066,249.312,-64.990,-177.329,7.302,148.597
C08578=1176.062,249.560,-65.017,-177.327,7.305,148.597
C08579=1176.058,249.809,-65.045,-177.324,7.306,148.597
C08580=1176.053,250.058,-65.072,-177.321,7.309,148.597
C08581=1176.049,250.306,-65.098,-177.319,7.312,148.597
C08582=1176.045,250.554,-65.125,-177.316,7.314,148.597
C08583=1176.040,250.803,-65.152,-177.313,7.317,148.596
C08584=1176.035,251.051,-65.180,-177.311,7.319,148.596
C08585=1176.031,251.299,-65.207,-177.308,7.322,148.596
C08586=1176.027,251.548,-65.235,-177.305,7.325,148.596
C08587=1176.023,251.797,-65.261,-177.303,7.327,148.596
C08588=1176.018,252.045,-65.288,-177.300,7.330,148.596
C08589=1176.014,252.294,-65.315,-177.297,7.333,148.596
C08590=1176.009,252.542,-65.342,-177.295,7.335,148.596
C08591=1176.004,252.791,-65.369,-177.292,7.338,148.595
C08592=1176.000,253.040,-65.397,-177.289,7.341,148.595
C08593=1175.996,253.288,-65.425,-177.287,7.343,148.595
C08594=1175.992,253.536,-65.451,-177.284,7.346,148.595
C08595=1175.987,253.784,-65.478,-177.282,7.348,148.595
C08596=1175.983,254.033,-65.505,-177.279,7.351,148.595
C08597=1175.979,254.282,-65.533,-177.276,7.354,148.595
C08598=1175.974,254.530,-65.560,-177.274,7.356,148.594
C08599=1175.970,254.778,-65.588,-177.271,7.359,148.594
C08600=1175.965,255.027,-65.615,-177.269,7.362,148.594
C08601=1175.960,255.275,-65.642,-177.266,7.363,148.594
C08602=1175.956,255.524,-65.670,-177.263,7.366,148.594
C08603=1175.952,255.773,-65.697,-177.260,7.369,148.594
C08604=1175.947,256.021,-65.724,-177.258,7.372,148.594
C08605=1175.943,256.269,-65.752,-177.255,7.374,148.594
C08606=1175.939,256.518,-65.779,-177.252,7.377,148.594
C08607=1175.934,256.767,-65.806,-177.250,7.379,148.593
C08608=1175.930,257.014,-65.834,-177.247,7.382,148.593
C08609=1175.925,257.263,-65.861,-177.245,7.385,148.593
C08610=1175.921,257.512,-65.889,-177.242,7.387,148.593
C08611=1175.917,257.760,-65.916,-177.240,7.390,148.593
C08612=1175.912,258.009,-65.943,-177.236,7.393,148.593
C08613=1175.908,258.256,-65.971,-177.234,7.395,148.593
C08614=1175.904,258.506,-65.998,-177.232,7.398,148.593
C08615=1175.899,258.753,-66.026,-177.229,7.401,148.593
C08616=1175.895,259.002,-66.053,-177.227,7.403,148.593
C08617=1175.891,259.251,-66.081,-177.224,7.406,148.593
C08618=1175.886,259.499,-66.109,-177.221,7.409,148.592
C08619=1175.882,259.747,-66.136,-177.219,7.411,148.592
C08620=1175.878,259.996,-66.164,-177.216,7.414,148.592
C08621=1175.873,260.244,-66.192,-177.213,7.417,148.592
C08622=1175.868,260.493,-66.219,-177.211,7.419,148.592
C08623=1175.864,260.741,-66.247,-177.208,7.422,148.592
C08624=1175.860,260.990,-66.274,-177.205,7.425,148.592
C08625=1175.855,261.238,-66.302,-177.202,7.428,148.592
C08626=1175.852,261.486,-66.330,-177.200,7.430,148.592
C08627=1175.847,261.735,-66.357,-177.197,7.433,148.591
C08628=1175.842,262.008,-66.388,-177.194,7.436,148.591
C08629=1175.837,262.281,-66.418,-177.192,7.439,148.591
C08630=1175.832,262.554,-66.449,-177.189,7.442,148.591
C08631=1175.828,262.827,-66.480,-177.186,7.444,148.591
C08632=1175.823,263.075,-66.507,-177.183,7.447,148.591
C08633=1175.818,263.323,-66.536,-177.180,7.450,148.591
C08634=1175.814,263.573,-66.563,-177.178,7.452,148.591
C08635=1175.810,263.821,-66.591,-177.175,7.455,148.591
C08636=1175.806,264.069,-66.619,-177.173,7.458,148.591
C08637=1175.801,264.318,-66.646,-177.170,7.461,148.591
C08638=1175.796,264.566,-66.675,-177.168,7.463,148.591
C08639=1175.793,264.814,-66.703,-177.165,7.466,148.590
C08640=1175.788,265.062,-66.731,-177.162,7.469,148.590
C08641=1175.784,265.311,-66.759,-177.160,7.471,148.590
C08642=1175.779,265.560,-66.786,-177.157,7.474,148.590
C08643=1175.775,265.808,-66.814,-177.154,7.477,148.590
C08644=1175.770,266.056,-66.843,-177.151,7.480,148.590
C08645=1175.766,266.304,-66.871,-177.149,7.482,148.590
C08646=1175.762,266.553,-66.899,-177.146,7.485,148.590
C08647=1175.757,266.801,-66.927,-177.144,7.488,148.590
C08648=1175.753,267.050,-66.955,-177.142,7.490,148.590
C08649=1175.749,267.298,-66.982,-177.139,7.493,148.590
C08650=1175.744,267.547,-67.011,-177.136,7.496,148.590
C08651=1175.740,267.795,-67.039,-177.133,7.499,148.590
C08652=1175.736,268.043,-67.067,-177.131,7.501,148.589
C08653=1175.731,268.292,-67.095,-177.128,7.504,148.589
C08654=1175.727,268.540,-67.124,-177.125,7.507,148.589
C08655=1175.722,268.788,-67.152,-177.122,7.510,148.589
C08656=1175.718,269.037,-67.180,-177.120,7.512,148.589
C08657=1175.714,269.285,-67.208,-177.118,7.515,148.589
C08658=1175.710,269.534,-67.237,-177.115,7.518,148.589
C08659=1175.705,269.782,-67.264,-177.112,7.521,148.589
C08660=1175.701,270.031,-67.293,-177.110,7.523,148.589
C08661=1175.696,270.278,-67.321,-177.107,7.526,148.589
C08662=1175.692,270.527,-67.350,-177.104,7.529,148.589
C08663=1175.688,270.775,-67.377,-177.102,7.532,148.589
C08664=1175.683,271.024,-67.406,-177.100,7.534,148.589
C08665=1175.679,271.272,-67.434,-177.097,7.537,148.589
C08666=1175.674,271.521,-67.463,-177.094,7.540,148.589
C08667=1175.670,271.768,-67.491,-177.091,7.543,148.589
C08668=1175.666,272.017,-67.520,-177.089,7.545,148.588
C08669=1175.662,272.266,-67.548,-177.086,7.548,148.588
C08670=1175.657,272.514,-67.576,-177.084,7.551,148.588
C08671=1175.653,272.762,-67.605,-177.081,7.554,148.588
C08672=1175.648,273.010,-67.633,-177.079,7.557,148.588
C08673=1175.645,273.258,-67.662,-177.076,7.560,148.588
C08674=1175.640,273.507,-67.690,-177.073,7.562,148.588
C08675=1175.636,273.755,-67.718,-177.071,7.565,148.588
C08676=1175.631,274.004,-67.747,-177.068,7.568,148.588
C08677=1175.627,274.251,-67.775,-177.066,7.571,148.588
C08678=1175.623,274.500,-67.804,-177.063,7.574,148.588
C08679=1175.618,274.749,-67.833,-177.060,7.577,148.588
C08680=1175.614,274.997,-67.861,-177.057,7.580,148.588
C08681=1175.610,275.245,-67.890,-177.055,7.582,148.588
C08682=1175.606,275.494,-67.918,-177.053,7.585,148.588
C08683=1175.601,275.742,-67.947,-177.050,7.588,148.588
C08684=1175.597,275.990,-67.976,-177.047,7.591,148.588
C08685=1175.592,276.238,-68.004,-177.044,7.594,148.588
C08686=1175.588,276.487,-68.033,-177.042,7.596,148.587
C08687=1175.584,276.735,-68.062,-177.039,7.599,148.587
C08688=1175.579,276.983,-68.090,-177.037,7.602,148.587
C08689=1175.575,277.231,-68.119,-177.034,7.605,148.587
C08690=1175.571,277.480,-68.148,-177.031,7.608,148.587
C08691=1175.567,277.729,-68.176,-177.029,7.610,148.587
C08692=1175.562,277.976,-68.205,-177.026,7.613,148.587
C08693=1175.558,278.225,-68.234,-177.024,7.616,148.587
C08694=1175.553,278.474,-68.264,-177.021,7.619,148.587
C08695=1175.549,278.722,-68.291,-177.018,7.622,148.587
C08696=1175.545,278.970,-68.321,-177.016,7.624,148.587
C08697=1175.540,279.219,-68.349,-177.013,7.627,148.587
C08698=1175.536,279.467,-68.379,-177.010,7.630,148.587
C08699=1175.532,279.715,-68.407,-177.008,7.633,148.587
C08700=1175.528,279.963,-68.436,-177.005,7.636,148.587
C08701=1175.523,280.212,-68.465,-177.003,7.638,148.587
C08702=1175.518,280.460,-68.494,-177.001,7.641,148.587
C08703=1175.515,280.707,-68.523,-176.998,7.644,148.587
C08704=1175.510,280.956,-68.552,-176.995,7.647,148.587
C08705=1175.506,281.205,-68.581,-176.992,7.650,148.587
C08706=1175.501,281.453,-68.609,-176.990,7.653,148.587
C08707=1175.497,281.701,-68.639,-176.987,7.655,148.587
C08708=1175.493,281.949,-68.668,-176.985,7.658,148.587
C08709=1175.489,282.198,-68.696,-176.982,7.661,148.587
C08710=1175.485,282.446,-68.726,-176.979,7.664,148.587
C08711=1175.480,282.694,-68.755,-176.976,7.667,148.587
C08712=1175.476,282.942,-68.784,-176.974,7.669,148.586
C08713=1175.471,283.191,-68.813,-176.972,7.673,148.587
C08714=1175.467,283.439,-68.843,-176.969,7.676,148.587
C08715=1175.463,283.687,-68.872,-176.967,7.679,148.587
C08716=1175.458,283.936,-68.900,-176.964,7.682,148.587
C08717=1175.454,284.184,-68.930,-176.961,7.685,148.586
C08718=1175.450,284.432,-68.959,-176.959,7.687,148.586
C08719=1175.445,284.680,-68.989,-176.956,7.690,148.586
C08720=1175.442,284.928,-69.018,-176.953,7.693,148.586
C08721=1175.437,285.177,-69.046,-176.951,7.696,148.586
C08722=1175.433,285.425,-69.076,-176.948,7.699,148.586
C08723=1175.429,285.673,-69.105,-176.946,7.702,148.586
C08724=1175.424,285.921,-69.134,-176.943,7.705,148.586
C08725=1175.420,286.170,-69.164,-176.941,7.707,148.586
C08726=1175.416,286.418,-69.193,-176.938,7.710,148.586
C08727=1175.412,286.666,-69.223,-176.935,7.713,148.586
C08728=1175.407,286.914,-69.252,-176.933,7.716,148.586
C08729=1175.403,287.163,-69.281,-176.930,7.719,148.586
C08730=1175.398,287.411,-69.310,-176.928,7.722,148.586
C08731=1175.394,287.659,-69.340,-176.925,7.724,148.586
C08732=1175.390,287.934,-69.373,-176.922,7.728,148.586
C08733=1175.384,288.209,-69.405,-176.919,7.731,148.586
C08734=1175.380,288.483,-69.438,-176.917,7.734,148.586
C08735=1175.375,288.758,-69.470,-176.913,7.738,148.586
C08736=1175.371,289.007,-69.500,-176.911,7.740,148.586
C08737=1175.367,289.255,-69.529,-176.908,7.743,148.586
C08738=1175.363,289.503,-69.559,-176.906,7.746,148.586
C08739=1175.358,289.751,-69.588,-176.903,7.749,148.586
C08740=1175.353,289.999,-69.618,-176.901,7.752,148.586
C08741=1175.349,290.247,-69.648,-176.898,7.755,148.586
C08742=1175.345,290.495,-69.678,-176.895,7.758,148.586
C08743=1175.341,290.744,-69.707,-176.893,7.761,148.586
C08744=1175.337,290.992,-69.736,-176.890,7.764,148.586
C08745=1175.332,291.240,-69.766,-176.888,7.766,148.586
C08746=1175.328,291.488,-69.795,-176.885,7.770,148.586
C08747=1175.323,291.737,-69.825,-176.883,7.773,148.586
C08748=1175.319,291.985,-69.856,-176.880,7.776,148.586
C08749=1175.315,292.233,-69.885,-176.877,7.779,148.586
C08750=1175.311,292.481,-69.914,-176.874,7.782,148.586
C08751=1175.307,292.729,-69.944,-176.872,7.785,148.586
C08752=1175.302,292.978,-69.974,-176.870,7.787,148.586
C08753=1175.298,293.226,-70.004,-176.867,7.790,148.586
C08754=1175.294,293.474,-70.034,-176.864,7.793,148.586
C08755=1175.290,293.722,-70.063,-176.862,7.796,148.586
C08756=1175.285,293.971,-70.093,-176.859,7.799,148.586
C08757=1175.281,294.218,-70.123,-176.857,7.802,148.586
C08758=1175.277,294.467,-70.153,-176.854,7.805,148.586
C08759=1175.272,294.715,-70.182,-176.851,7.808,148.586
C08760=1175.268,294.963,-70.213,-176.849,7.811,148.586
C08761=1175.264,295.211,-70.242,-176.847,7.814,148.586
C08762=1175.260,295.459,-70.272,-176.844,7.817,148.586
C08763=1175.256,295.707,-70.302,-176.841,7.820,148.586
C08764=1175.251,295.956,-70.332,-176.839,7.823,148.586
C08765=1175.247,296.204,-70.363,-176.836,7.826,148.586
C08766=1175.243,296.452,-70.392,-176.834,7.829,148.586
C08767=1175.238,296.701,-70.422,-176.831,7.832,148.586
C08768=1175.234,296.949,-70.452,-176.828,7.835,148.586
C08769=1175.230,297.197,-70.482,-176.825,7.838,148.586
C08770=1175.226,297.445,-70.512,-176.823,7.841,148.587
C08771=1175.221,297.693,-70.542,-176.821,7.843,148.586
C08772=1175.217,297.941,-70.573,-176.818,7.846,148.586
C08773=1175.213,298.189,-70.602,-176.816,7.849,148.586
C08774=1175.209,298.437,-70.632,-176.813,7.853,148.587
C08775=1175.204,298.686,-70.663,-176.810,7.856,148.587
C08776=1175.201,298.934,-70.693,-176.808,7.859,148.587
C08777=1175.196,299.182,-70.724,-176.805,7.862,148.586
C08778=1175.192,299.430,-70.753,-176.803,7.865,148.587
C08779=1175.187,299.678,-70.784,-176.800,7.868,148.587
C08780=1175.183,299.926,-70.813,-176.797,7.871,148.587
C08781=1175.179,300.174,-70.843,-176.795,7.874,148.587
C08782=1175.175,300.422,-70.874,-176.793,7.876,148.587
C08783=1175.171,300.671,-70.904,-176.790,7.879,148.587
C08784=1175.166,300.919,-70.935,-176.787,7.882,148.587
C08785=1175.162,301.166,-70.965,-176.785,7.885,148.587
C08786=1175.158,301.415,-70.995,-176.782,7.889,148.587
C08787=1175.154,301.663,-71.025,-176.780,7.892,148.587
C08788=1175.150,301.911,-71.056,-176.777,7.895,148.587
C08789=1175.145,302.160,-71.086,-176.775,7.898,148.587
C08790=1175.141,302.408,-71.117,-176.772,7.901,148.587
C08791=1175.136,302.655,-71.147,-176.769,7.904,148.587
C08792=1175.132,302.903,-71.178,-176.766,7.907,148.587
C08793=1175.127,303.152,-71.208,-176.764,7.910,148.587
C08794=1175.124,303.400,-71.238,-176.761,7.913,148.587
C08795=1175.120,303.648,-71.269,-176.759,7.916,148.587
C08796=1175.115,303.896,-71.300,-176.756,7.919,148.587
C08797=1175.111,304.144,-71.330,-176.754,7.922,148.587
C08798=1175.107,304.393,-71.360,-176.752,7.925,148.587
C08799=1175.103,304.641,-71.390,-176.749,7.928,148.587
C08800=1175.098,304.889,-71.421,-176.747,7.931,148.587
C08801=1175.094,305.136,-71.452,-176.744,7.934,148.587
C08802=1175.090,305.384,-71.482,-176.742,7.937,148.588
C08803=1175.086,305.633,-71.513,-176.739,7.940,148.587
C08804=1175.081,305.881,-71.544,-176.736,7.943,148.587
C08805=1175.077,306.128,-71.574,-176.734,7.946,148.588
C08806=1175.073,306.377,-71.605,-176.731,7.949,148.588
C08807=1175.069,306.625,-71.636,-176.728,7.952,148.588
C08808=1175.065,306.873,-71.666,-176.726,7.956,148.588
C08809=1175.060,307.121,-71.697,-176.723,7.959,148.588
C08810=1175.056,307.369,-71.728,-176.721,7.962,148.588
C08811=1175.052,307.617,-71.759,-176.718,7.965,148.588
C08812=1175.048,307.865,-71.789,-176.716,7.968,148.588
C08813=1175.044,308.114,-71.820,-176.713,7.971,148.588
C08814=1175.039,308.361,-71.851,-176.711,7.974,148.588
C08815=1175.034,308.609,-71.882,-176.708,7.977,148.588
C08816=1175.031,308.857,-71.912,-176.705,7.980,148.588
C08817=1175.027,309.106,-71.943,-176.703,7.984,148.588
C08818=1175.022,309.354,-71.974,-176.700,7.987,148.588
C08819=1175.017,309.602,-72.005,-176.698,7.989,148.588
C08820=1175.014,309.850,-72.035,-176.696,7.992,148.588
C08821=1175.009,310.098,-72.066,-176.693,7.995,148.588
C08822=1175.006,310.346,-72.098,-176.691,7.998,148.589
C08823=1175.001,310.594,-72.128,-176.688,8.001,148.589
C08824=1174.997,310.842,-72.159,-176.685,8.004,148.589
C08825=1174.992,311.091,-72.190,-176.683,8.008,148.589
C08826=1174.989,311.338,-72.220,-176.680,8.011,148.589
C08827=1174.984,311.586,-72.252,-176.678,8.014,148.589
C08828=1174.980,311.834,-72.283,-176.675,8.017,148.589
C08829=1174.976,312.082,-72.314,-176.673,8.020,148.589
C08830=1174.972,312.331,-72.345,-176.670,8.023,148.589
C08831=1174.967,312.578,-72.376,-176.668,8.026,148.589
C08832=1174.963,312.826,-72.407,-176.665,8.029,148.589
C08833=1174.959,313.075,-72.438,-176.663,8.032,148.589
C08834=1174.955,313.322,-72.469,-176.660,8.035,148.589
C08835=1174.951,313.570,-72.500,-176.658,8.039,148.589
C08836=1174.946,313.847,-72.536,-176.654,8.043,148.589
C08837=1174.942,314.124,-72.570,-176.652,8.046,148.590
C08838=1174.937,314.401,-72.605,-176.649,8.049,148.590
C08839=1174.932,314.678,-72.640,-176.646,8.053,148.590
C08840=1174.927,314.926,-72.671,-176.644,8.056,148.590
C08841=1174.923,315.173,-72.702,-176.641,8.059,148.590
C08842=1174.919,315.422,-72.733,-176.639,8.062,148.590
C08843=1174.914,315.670,-72.764,-176.636,8.065,148.590
C08844=1174.911,315.918,-72.796,-176.633,8.068,148.590
C08845=1174.906,316.166,-72.827,-176.631,8.071,148.590
C08846=1174.902,316.414,-72.859,-176.628,8.074,148.590
C08847=1174.898,316.662,-72.889,-176.626,8.078,148.590
C08848=1174.894,316.910,-72.921,-176.623,8.081,148.590
C08849=1174.889,317.158,-72.952,-176.621,8.084,148.591
C08850=1174.886,317.406,-72.984,-176.618,8.087,148.591
C08851=1174.881,317.654,-73.015,-176.616,8.090,148.591
C08852=1174.877,317.902,-73.046,-176.613,8.093,148.591
C08853=1174.873,318.149,-73.078,-176.611,8.097,148.591
C08854=1174.869,318.398,-73.109,-176.608,8.100,148.591
C08855=1174.865,318.645,-73.141,-176.606,8.103,148.591
C08856=1174.861,318.894,-73.172,-176.603,8.106,148.591
C08857=1174.857,319.142,-73.203,-176.601,8.109,148.591
C08858=1174.853,319.389,-73.235,-176.598,8.112,148.591
C08859=1174.849,319.638,-73.266,-176.596,8.116,148.591
C08860=1174.844,319.886,-73.298,-176.593,8.119,148.591
C08861=1174.840,320.134,-73.330,-176.591,8.122,148.592
C08862=1174.835,320.382,-73.361,-176.588,8.125,148.592
C08863=1174.832,320.630,-73.393,-176.586,8.128,148.592
C08864=1174.827,320.877,-73.424,-176.583,8.131,148.592
C08865=1174.824,321.125,-73.456,-176.581,8.134,148.592
C08866=1174.819,321.374,-73.488,-176.578,8.137,148.592
C08867=1174.815,321.621,-73.519,-176.576,8.141,148.592
C08868=1174.811,321.869,-73.551,-176.573,8.144,148.592
C08869=1174.807,322.117,-73.582,-176.571,8.147,148.592
C08870=1174.803,322.365,-73.614,-176.568,8.150,148.592
C08871=1174.798,322.614,-73.646,-176.566,8.153,148.593
C08872=1174.794,322.861,-73.678,-176.563,8.156,148.593
C08873=1174.790,323.109,-73.709,-176.561,8.160,148.593
C08874=1174.786,323.357,-73.741,-176.558,8.163,148.593
C08875=1174.781,323.605,-73.773,-176.556,8.166,148.593
C08876=1174.778,323.853,-73.805,-176.554,8.169,148.593
C08877=1174.774,324.101,-73.837,-176.551,8.172,148.593
C08878=1174.770,324.348,-73.868,-176.548,8.176,148.593
C08879=1174.765,324.597,-73.901,-176.545,8.179,148.593
C08880=1174.761,324.845,-73.932,-176.543,8.183,148.594
C08881=1174.757,325.093,-73.964,-176.540,8.186,148.594
C08882=1174.752,325.341,-73.996,-176.538,8.189,148.594
C08883=1174.749,325.589,-74.028,-176.536,8.192,148.594
C08884=1174.744,325.836,-74.059,-176.533,8.195,148.594
C08885=1174.740,326.085,-74.092,-176.531,8.198,148.594
C08886=1174.736,326.333,-74.124,-176.528,8.201,148.594
C08887=1174.732,326.580,-74.155,-176.526,8.205,148.594
C08888=1174.728,326.828,-74.187,-176.523,8.208,148.595
C08889=1174.724,327.076,-74.220,-176.521,8.211,148.595
C08890=1174.720,327.323,-74.252,-176.518,8.214,148.595
C08891=1174.715,327.572,-74.284,-176.516,8.217,148.595
C08892=1174.712,327.820,-74.316,-176.513,8.221,148.595
C08893=1174.707,328.068,-74.348,-176.511,8.224,148.595
C08894=1174.703,328.315,-74.380,-176.508,8.227,148.595
C08895=1174.699,328.563,-74.412,-176.506,8.230,148.595
C08896=1174.695,328.812,-74.444,-176.504,8.234,148.596
C08897=1174.691,329.058,-74.476,-176.501,8.237,148.596
C08898=1174.686,329.307,-74.509,-176.498,8.241,148.596
C08899=1174.683,329.555,-74.541,-176.496,8.244,148.596
C08900=1174.678,329.803,-74.573,-176.493,8.247,148.596
C08901=1174.674,330.050,-74.604,-176.491,8.250,148.596
C08902=1174.670,330.298,-74.638,-176.488,8.253,148.596
C08903=1174.666,330.546,-74.669,-176.486,8.257,148.597
C08904=1174.662,330.795,-74.702,-176.484,8.260,148.597
C08905=1174.658,331.043,-74.734,-176.482,8.263,148.597
C08906=1174.653,331.290,-74.767,-176.479,8.266,148.597
C08907=1174.649,331.538,-74.798,-176.477,8.269,148.597
C08908=1174.645,331.786,-74.831,-176.474,8.273,148.597
C08909=1174.642,332.033,-74.863,-176.472,8.276,148.597
C08910=1174.637,332.282,-74.896,-176.469,8.279,148.598
C08911=1174.632,332.529,-74.928,-176.467,8.282,148.598
C08912=1174.629,332.777,-74.960,-176.464,8.286,148.598
C08913=1174.624,333.025,-74.993,-176.461,8.290,148.598
C08914=1174.621,333.273,-75.025,-176.459,8.293,148.598
C08915=1174.616,333.521,-75.058,-176.457,8.296,148.598
C08916=1174.611,333.769,-75.090,-176.454,8.299,148.598
C08917=1174.608,334.016,-75.123,-176.452,8.302,148.599
C08918=1174.603,334.264,-75.155,-176.450,8.306,148.599
C08919=1174.600,334.512,-75.188,-176.447,8.309,148.599
C08920=1174.596,334.760,-75.220,-176.445,8.312,148.599
C08921=1174.592,335.008,-75.253,-176.442,8.315,148.599
C08922=1174.588,335.256,-75.285,-176.440,8.319,148.599
C08923=1174.584,335.504,-75.318,-176.438,8.322,148.600
C08924=1174.579,335.751,-75.350,-176.434,8.326,148.600
C08925=1174.575,335.999,-75.383,-176.432,8.329,148.600
C08926=1174.571,336.247,-75.415,-176.430,8.332,148.600
C08927=1174.567,336.495,-75.448,-176.428,8.336,148.600
C08928=1174.562,336.743,-75.481,-176.425,8.339,148.600
C08929=1174.559,336.991,-75.513,-176.423,8.342,148.601
C08930=1174.555,337.238,-75.546,-176.420,8.345,148.601
C08931=1174.550,337.487,-75.579,-176.418,8.349,148.601
C08932=1174.547,337.734,-75.611,-176.416,8.352,148.601
C08933=1174.543,337.982,-75.645,-176.413,8.355,148.601
C08934=1174.538,338.230,-75.677,-176.410,8.359,148.601
C08935=1174.533,338.477,-75.710,-176.408,8.362,148.602
C08936=1174.529,338.725,-75.743,-176.406,8.366,148.602
C08937=1174.526,338.973,-75.775,-176.403,8.369,148.602
C08938=1174.522,339.221,-75.808,-176.401,8.372,148.602
C08939=1174.517,339.468,-75.841,-176.398,8.375,148.602
C08940=1174.514,339.748,-75.878,-176.396,8.379,148.603
C08941=1174.508,340.027,-75.915,-176.393,8.383,148.603
C08942=1174.503,340.307,-75.952,-176.390,8.387,148.603
C08943=1174.499,340.585,-75.989,-176.388,8.391,148.603
C08944=1174.495,340.833,-76.022,-176.385,8.394,148.603
C08945=1174.491,341.081,-76.055,-176.383,8.398,148.604
C08946=1174.487,341.328,-76.088,-176.380,8.401,148.604
C08947=1174.482,341.576,-76.121,-176.378,8.404,148.604
C08948=1174.478,341.825,-76.154,-176.376,8.407,148.604
C08949=1174.474,342.072,-76.187,-176.374,8.410,148.604
C08950=1174.470,342.320,-76.220,-176.371,8.415,148.605
C08951=1174.466,342.568,-76.253,-176.368,8.418,148.605
C08952=1174.461,342.815,-76.286,-176.366,8.421,148.605
C08953=1174.458,343.063,-76.319,-176.364,8.424,148.605
C08954=1174.454,343.311,-76.352,-176.362,8.428,148.605
C08955=1174.450,343.558,-76.385,-176.359,8.431,148.606
C08956=1174.446,343.807,-76.419,-176.357,8.434,148.606
C08957=1174.442,344.055,-76.452,-176.355,8.438,148.606
C08958=1174.438,344.302,-76.485,-176.352,8.442,148.606
C08959=1174.434,344.550,-76.518,-176.350,8.445,148.607
C08960=1174.430,344.798,-76.551,-176.347,8.448,148.607
C08961=1174.425,345.045,-76.585,-176.345,8.451,148.607
C08962=1174.421,345.293,-76.618,-176.342,8.455,148.607
C08963=1174.417,345.541,-76.651,-176.340,8.458,148.607
C08964=1174.413,345.789,-76.684,-176.338,8.461,148.607
C08965=1174.409,346.036,-76.717,-176.335,8.465,148.608
C08966=1174.405,346.284,-76.750,-176.333,8.469,148.608
C08967=1174.401,346.532,-76.783,-176.330,8.472,148.608
C08968=1174.396,346.780,-76.817,-176.328,8.475,148.608
C08969=1174.392,347.027,-76.851,-176.326,8.479,148.609
C08970=1174.388,347.275,-76.885,-176.324,8.482,148.609
C08971=1174.384,347.523,-76.918,-176.321,8.486,148.609
C08972=1174.380,347.771,-76.951,-176.319,8.490,148.609
C08973=1174.376,348.019,-76.984,-176.317,8.493,148.610
C08974=1174.372,348.266,-77.018,-176.314,8.496,148.610
C08975=1174.368,348.513,-77.051,-176.312,8.500,148.610
C08976=1174.364,348.761,-77.084,-176.310,8.503,148.610
C08977=1174.360,349.010,-77.118,-176.307,8.507,148.611
C08978=1174.356,349.257,-77.152,-176.305,8.510,148.611
C08979=1174.352,349.505,-77.185,-176.302,8.514,148.611
C08980=1174.348,349.752,-77.219,-176.300,8.517,148.611
C08981=1174.343,350.000,-77.252,-176.298,8.520,148.611
C08982=1174.340,350.247,-77.286,-176.296,8.524,148.612
C08983=1174.336,350.496,-77.319,-176.293,8.528,148.612
C08984=1174.331,350.744,-77.353,-176.291,8.531,148.612
C08985=1174.327,350.991,-77.387,-176.289,8.535,148.613
C08986=1174.323,351.239,-77.420,-176.286,8.538,148.613
C08987=1174.319,351.486,-77.454,-176.284,8.541,148.613
C08988=1174.316,351.734,-77.487,-176.282,8.545,148.613
C08989=1174.311,351.982,-77.521,-176.279,8.549,148.614
C08990=1174.307,352.229,-77.555,-176.277,8.552,148.614
C08991=1174.303,352.477,-77.588,-176.275,8.556,148.614
C08992=1174.299,352.724,-77.622,-176.273,8.559,148.614
C08993=1174.295,352.973,-77.656,-176.270,8.562,148.615
C08994=1174.291,353.220,-77.690,-176.268,8.567,148.615
C08995=1174.287,353.468,-77.723,-176.266,8.570,148.615
C08996=1174.282,353.715,-77.758,-176.263,8.573,148.615
C08997=1174.279,353.964,-77.791,-176.261,8.577,148.616
C08998=1174.275,354.211,-77.825,-176.259,8.580,148.616
C08999=1174.271,354.458,-77.858,-176.256,8.584,148.616
C09000=1174.266,354.706,-77.893,-176.254,8.588,148.617
C09001=1174.263,354.954,-77.926,-176.252,8.591,148.617
C09002=1174.259,355.201,-77.960,-176.250,8.594,148.617
C09003=1174.254,355.449,-77.994,-176.248,8.598,148.617
C09004=1174.251,355.697,-78.028,-176.245,8.602,148.618
C09005=1174.246,355.945,-78.062,-176.243,8.605,148.618
C09006=1174.242,356.192,-78.096,-176.241,8.609,148.618
C09007=1174.238,356.439,-78.129,-176.238,8.612,148.619
C09008=1174.234,356.688,-78.164,-176.236,8.615,148.619
C09009=1174.230,356.935,-78.198,-176.234,8.620,148.619
C09010=1174.226,357.182,-78.231,-176.232,8.623,148.620
C09011=1174.222,357.431,-78.266,-176.229,8.627,148.620
C09012=1174.218,357.678,-78.300,-176.227,8.630,148.620
C09013=1174.214,357.926,-78.334,-176.225,8.634,148.620
C09014=1174.210,358.173,-78.368,-176.222,8.638,148.621
C09015=1174.206,358.421,-78.402,-176.220,8.641,148.621
C09016=1174.202,358.668,-78.436,-176.218,8.644,148.621
C09017=1174.198,358.916,-78.470,-176.216,8.648,148.622
C09018=1174.194,359.164,-78.504,-176.213,8.652,148.622
C09019=1174.190,359.411,-78.538,-176.211,8.656,148.622
C09020=1174.186,359.659,-78.573,-176.209,8.659,148.623
C09021=1174.182,359.906,-78.607,-176.207,8.662,148.623
C09022=1174.178,360.154,-78.642,-176.205,8.666,148.623
C09023=1174.174,360.401,-78.676,-176.202,8.670,148.624
C09024=1174.170,360.649,-78.709,-176.201,8.674,148.624
C09025=1174.166,360.897,-78.744,-176.198,8.677,148.624
C09026=1174.162,361.145,-78.778,-176.196,8.681,148.625
C09027=1174.159,361.393,-78.812,-176.195,8.684,148.625
C09028=1174.154,361.640,-78.847,-176.192,8.688,148.625
C09029=1174.149,361.887,-78.881,-176.190,8.692,148.626
C09030=1174.146,362.135,-78.915,-176.188,8.695,148.626
C09031=1174.142,362.383,-78.950,-176.186,8.699,148.626
C09032=1174.138,362.630,-78.984,-176.184,8.703,148.627
C09033=1174.134,362.878,-79.019,-176.181,8.707,148.627
C09034=1174.131,363.126,-79.053,-176.179,8.710,148.628
C09035=1174.126,363.373,-79.087,-176.177,8.714,148.628
C09036=1174.122,363.621,-79.122,-176.175,8.717,148.628
C09037=1174.118,363.868,-79.156,-176.173,8.721,148.629
C09038=1174.114,364.116,-79.190,-176.172,8.724,148.629
C09039=1174.110,364.364,-79.225,-176.170,8.728,148.630
C09040=1174.106,364.611,-79.259,-176.167,8.732,148.630
C09041=1174.102,364.858,-79.295,-176.165,8.736,148.630
C09042=1174.098,365.106,-79.329,-176.163,8.739,148.631
C09043=1174.094,365.354,-79.363,-176.161,8.743,148.631
C09044=1174.089,365.635,-79.403,-176.159,8.747,148.632
C09045=1174.085,365.918,-79.443,-176.157,8.751,148.632
C09046=1174.081,366.200,-79.481,-176.155,8.756,148.632
C09047=1174.076,366.481,-79.520,-176.152,8.760,148.633
C09048=1174.072,366.729,-79.556,-176.150,8.764,148.633
C09049=1174.068,366.977,-79.591,-176.149,8.767,148.634
C09050=1174.064,367.224,-79.625,-176.147,8.771,148.634
C09051=1174.060,367.472,-79.659,-176.145,8.774,148.635
C09052=1174.056,367.719,-79.695,-176.143,8.778,148.635
C09053=1174.052,367.967,-79.729,-176.141,8.782,148.636
C09054=1174.048,368.214,-79.763,-176.139,8.785,148.636
C09055=1174.044,368.462,-79.798,-176.138,8.789,148.636
C09056=1174.040,368.709,-79.833,-176.136,8.792,148.637
C09057=1174.036,368.957,-79.868,-176.134,8.796,148.637
C09058=1174.032,369.205,-79.903,-176.132,8.800,148.638
C09059=1174.029,369.452,-79.938,-176.131,8.804,148.638
C09060=1174.024,369.699,-79.972,-176.129,8.807,148.639
C09061=1174.020,369.947,-80.007,-176.127,8.811,148.639
C09062=1174.016,370.195,-80.042,-176.126,8.815,148.640
C09063=1174.012,370.442,-80.077,-176.124,8.818,148.640
C09064=1174.008,370.690,-80.112,-176.122,8.822,148.641
C09065=1174.004,370.937,-80.146,-176.120,8.826,148.641
C09066=1174.000,371.185,-80.181,-176.119,8.829,148.642
C09067=1173.996,371.432,-80.216,-176.117,8.832,148.642
C09068=1173.992,371.680,-80.251,-176.116,8.836,148.643
C09069=1173.989,371.927,-80.287,-176.114,8.840,148.643
C09070=1173.984,372.175,-80.321,-176.113,8.844,148.644
C09071=1173.980,372.422,-80.357,-176.111,8.847,148.644
C09072=1173.976,372.670,-80.391,-176.109,8.851,148.645
C09073=1173.973,372.917,-80.426,-176.108,8.855,148.645
C09074=1173.969,373.165,-80.461,-176.107,8.858,148.646
C09075=1173.965,373.412,-80.496,-176.105,8.862,148.646
C09076=1173.961,373.660,-80.531,-176.104,8.865,148.647
C09077=1173.957,373.907,-80.567,-176.102,8.869,148.648
C09078=1173.952,374.155,-80.601,-176.101,8.872,148.648
C09079=1173.949,374.402,-80.637,-176.100,8.876,148.649
C09080=1173.945,374.650,-80.672,-176.098,8.880,148.649
C09081=1173.940,374.897,-80.707,-176.096,8.884,148.650
C09082=1173.937,375.145,-80.742,-176.095,8.887,148.650
C09083=1173.933,375.393,-80.777,-176.094,8.891,148.651
C09084=1173.929,375.640,-80.812,-176.092,8.894,148.651
C09085=1173.925,375.887,-80.848,-176.091,8.897,148.652
C09086=1173.921,376.135,-80.882,-176.090,8.901,148.652
C09087=1173.917,376.382,-80.918,-176.089,8.905,148.653
C09088=1173.913,376.630,-80.953,-176.088,8.908,148.654
C09089=1173.909,376.878,-80.988,-176.086,8.912,148.654
C09090=1173.905,377.125,-81.023,-176.085,8.915,148.655
C09091=1173.901,377.372,-81.059,-176.084,8.919,148.655
C09092=1173.897,377.620,-81.094,-176.082,8.923,148.656
C09093=1173.893,377.867,-81.129,-176.081,8.926,148.657
C09094=1173.889,378.114,-81.164,-176.080,8.930,148.657
C09095=1173.886,378.362,-81.200,-176.079,8.933,148.658
C09096=1173.881,378.609,-81.234,-176.078,8.937,148.658
C09097=1173.877,378.857,-81.270,-176.077,8.940,148.659
C09098=1173.874,379.104,-81.305,-176.076,8.943,148.660
C09099=1173.870,379.352,-81.341,-176.075,8.947,148.660
C09100=1173.865,379.599,-81.375,-176.074,8.950,148.661
C09101=1173.862,379.847,-81.411,-176.073,8.954,148.662
C09102=1173.858,380.094,-81.447,-176.072,8.957,148.662
C09103=1173.853,380.341,-81.482,-176.071,8.960,148.663
C09104=1173.849,380.589,-81.518,-176.070,8.964,148.663
C09105=1173.845,380.837,-81.553,-176.069,8.967,148.664
C09106=1173.842,381.085,-81.588,-176.069,8.971,148.665
C09107=1173.838,381.331,-81.623,-176.067,8.975,148.665
C09108=1173.834,381.579,-81.659,-176.066,8.978,148.666
C09109=1173.830,381.826,-81.695,-176.065,8.981,148.666
C09110=1173.827,382.074,-81.730,-176.065,8.984,148.667
C09111=1173.822,382.321,-81.766,-176.064,8.988,148.668
C09112=1173.818,382.569,-81.801,-176.063,8.991,148.668
C09113=1173.814,382.817,-81.836,-176.062,8.995,148.669
C09114=1173.810,383.064,-81.872,-176.062,8.998,148.670
C09115=1173.806,383.311,-81.907,-176.061,9.001,148.671
C09116=1173.802,383.558,-81.943,-176.060,9.004,148.671
C09117=1173.799,383.806,-81.978,-176.059,9.007,148.672
C09118=1173.794,384.054,-82.014,-176.059,9.011,148.673
C09119=1173.791,384.301,-82.050,-176.058,9.014,148.673
C09120=1173.786,384.548,-82.085,-176.058,9.017,148.674
C09121=1173.783,384.795,-82.120,-176.057,9.020,148.674
C09122=1173.779,385.043,-82.156,-176.057,9.024,148.675
C09123=1173.775,385.291,-82.192,-176.056,9.027,148.676
C09124=1173.770,385.538,-82.227,-176.055,9.030,148.677
C09125=1173.767,385.785,-82.263,-176.054,9.033,148.677
C09126=1173.763,386.033,-82.298,-176.054,9.037,148.678
C09127=1173.759,386.280,-82.334,-176.054,9.040,148.679
C09128=1173.755,386.528,-82.370,-176.053,9.043,148.679
C09129=1173.751,386.775,-82.406,-176.053,9.046,148.680
C09130=1173.747,387.022,-82.441,-176.053,9.049,148.681
C09131=1173.743,387.270,-82.476,-176.052,9.052,148.681
C09132=1173.739,387.518,-82.513,-176.051,9.056,148.682
C09133=1173.735,387.765,-82.548,-176.052,9.058,148.683
C09134=1173.732,388.013,-82.584,-176.051,9.061,148.683
C09135=1173.727,388.259,-82.619,-176.050,9.065,148.684
C09136=1173.724,388.507,-82.654,-176.050,9.067,148.685
C09137=1173.719,388.755,-82.691,-176.050,9.070,148.685
C09138=1173.716,389.001,-82.727,-176.049,9.074,148.686
C09139=1173.712,389.249,-82.762,-176.049,9.076,148.687
C09140=1173.708,389.497,-82.798,-176.049,9.080,148.688
C09141=1173.704,389.744,-82.834,-176.049,9.082,148.688
C09142=1173.700,389.991,-82.869,-176.048,9.085,148.689
C09143=1173.696,390.239,-82.905,-176.048,9.088,148.690
